	IF NOT #MovementActive THEN
	    FOR #i := 0 TO 12 DO
	        IF #ProductBuffer[#i].Active THEN
	            // Distance is oriented by DirectionSign:
	            //  - If DirectionSign = +1: Distance = Encoder - Start  (forward positive)
	            //  - If DirectionSign = -1: Distance = Start   - Encoder (forward negative)
	            #Distance := #DirectionSign * (#EncoderPosition - #ProductBuffer[#i].StartPosition);
	            
	            IF #Distance >= #TriggerDistance THEN
	                #TriggerMovement := TRUE;
	                #MovementActive := TRUE;
	                #ProductBuffer[#i].Active := FALSE;
	                EXIT;
	            END_IF;
	        END_IF;
	    END_FOR;
	END_IF;
	
	
	// 4️⃣ Wacht op feedback om beweging af te ronden
	IF #MovementActive AND #TriggerFeedback THEN
	    #TriggerMovement := FALSE;
	    #MovementActive := FALSE;
	END_IF;
	
END_FUNCTION_BLOCK

FUNCTION_BLOCK "BlowOff_Timer"
{ S7_Optimized_Access := 'FALSE' }
VERSION : 0.1
   VAR_INPUT 
      Enable : Bool;
      CycleTime : Time;
      PulseDuration : Time;
      NowTime : Time;
   END_VAR

   VAR_OUTPUT 
      Q_Pulse : Bool;
   END_VAR

   VAR 
      CycleTimer {InstructionName := 'TON'; LibVersion := '1.0'; S7_SetPoint := 'False'} : TON;
      PulseTimer {InstructionName := 'TON'; LibVersion := '1.0'; S7_SetPoint := 'False'} : TON;
      State { S7_SetPoint := 'True'} : Int;
      S_PEXT : Int;
   END_VAR

   VAR_TEMP 
      PulseActive : Bool;
      StartPulse : Bool;
      TriggerPulse : Bool;
      PulseBusy : Bool;
      DummyWord : Word;
      DummyWord2 : Bool;
      T1 : Int;
      PulseStartTime : Time;
      LastPulseEndTime : Time;
      LastPulseTime : Time;
   END_VAR


BEGIN
	// Logica
	IF #Enable THEN
	    // Start cyclische timer
	    #CycleTimer(IN := TRUE,
	                PT := #CycleTime);
	    
	    IF #CycleTimer.Q THEN
	        // Start puls-timer als cyclus voorbij is
	        #PulseTimer(IN := TRUE,
	                    PT := #PulseDuration);
	        
	        // Reset de CycleTimer voor de volgende cyclus
	        #CycleTimer(IN := FALSE,
	                    PT := #CycleTime);
	    END_IF;
	    
	    // Puls-timer logica
	    IF #PulseTimer.IN THEN
	        #Q_Pulse := TRUE;
	        
	        IF #PulseTimer.Q THEN
	            // Puls voorbij, pulse output uit
	            #PulseTimer(IN := FALSE,
	                        PT := #PulseDuration);
	            #Q_Pulse := FALSE;
	        END_IF;
	    ELSE
	        #Q_Pulse := FALSE;
	    END_IF;
	    
	ELSE
	    // Alles resetten bij disable
	    #CycleTimer(IN := FALSE,
	                PT := #CycleTime);
	    #PulseTimer(IN := FALSE,
	                PT := #PulseDuration);
	    #Q_Pulse := FALSE;
	END_IF;
	
END_FUNCTION_BLOCK

FUNCTION "4 - Prog. 2" : Void   // FC2, LAD
TITLE = System Program 2
VERSION : 0.1
// stored: AutoNumber true, IsIECCheckEnabled false, UDAEnableTagReadback false
   VAR_TEMP
      Retourband_Delayed : Bool;
      BlowOffTimer : Bool;
      Democoil : Bool;
      StartBlowOff : Bool;
      Pos2_Done : Bool;
      BlowOff_Activated : Bool;
      AandrukCilindersOut : Bool;
      Move2Busy : Bool;
      ProductBehindWals : Bool;
      SR_Move2 : Bool;
      Move1Busy : Bool;
   END_VAR
   VAR_TEMP   // added for the SCL form of the ladder/FBD networks
      _w1 : Bool;
   END_VAR
BEGIN

REGION Network 1: Close 1 Magazine Hole (cilinder)
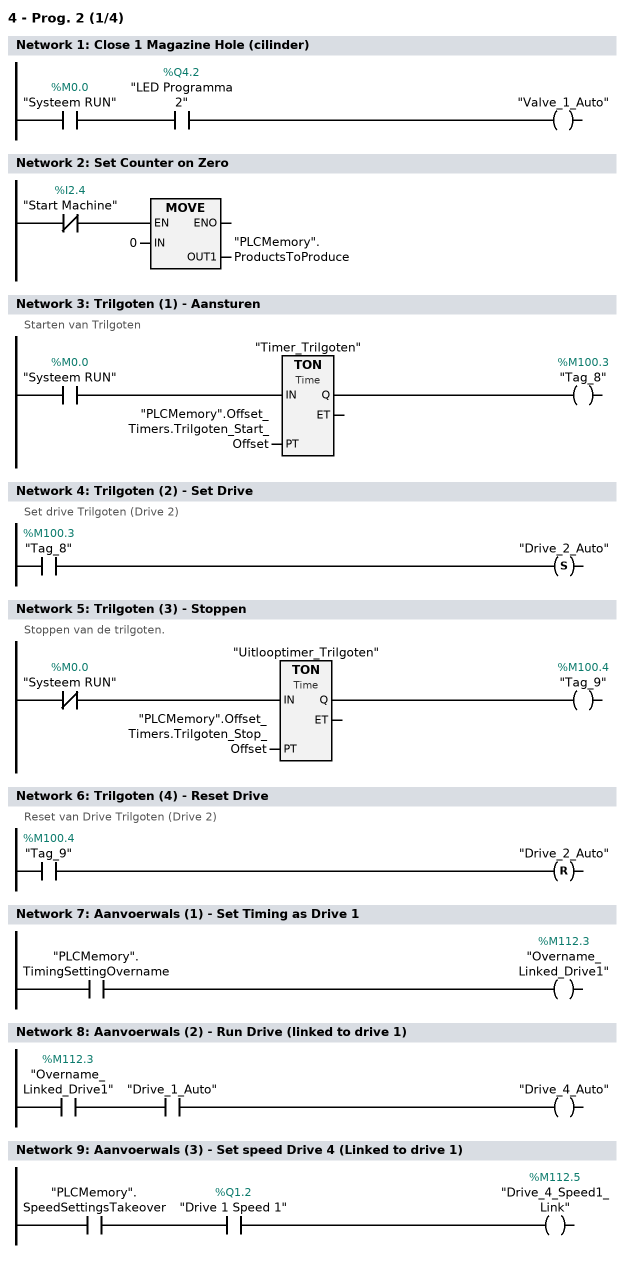
   RUNG wire#powerrail
      Contact( "Systeem RUN" )
      Contact( "LED Programma 2" )
      Coil( "Valve_1_Auto" )
   END_RUNG
   // the same network as SCL:
   "Valve_1_Auto" := "Systeem RUN" AND "LED Programma 2";
END_REGION

REGION Network 2: Set Counter on Zero
   RUNG wire#powerrail
      I_Contact( "Start Machine" )
      { S7_GenerateENO := "TRUE" } Move(in := 0, out1 => "PLCMemory".ProductsToProduce)
   END_RUNG
   // the same network as SCL:
   IF NOT "Start Machine" THEN "PLCMemory".ProductsToProduce := 0; END_IF;
END_REGION

REGION Network 3: Trilgoten (1) - Aansturen
   // Starten van Trilgoten
   RUNG wire#powerrail
      Contact( "Systeem RUN" )
      { S7_Templates := "time_type := Time" } "Timer_Trilgoten".TON(pt := "PLCMemory".Offset_Timers.Trilgoten_Start_Offset, et =>)
      Coil( "Tag_8" )
   END_RUNG
   // the same network as SCL:
   "Timer_Trilgoten".TON(IN := "Systeem RUN", PT := "PLCMemory".Offset_Timers.Trilgoten_Start_Offset);
   "Tag_8" := "Timer_Trilgoten".Q;
END_REGION

REGION Network 4: Trilgoten (2) - Set Drive
   // Set drive Trilgoten (Drive 2)
   RUNG wire#powerrail
      Contact( "Tag_8" )
      S_Coil( "Drive_2_Auto" )
   END_RUNG
   // the same network as SCL:
   IF "Tag_8" THEN "Drive_2_Auto" := TRUE; END_IF;
END_REGION

REGION Network 5: Trilgoten (3) - Stoppen
   // Stoppen van de trilgoten.
   RUNG wire#powerrail
      I_Contact( "Systeem RUN" )
      { S7_Templates := "time_type := Time" } "Uitlooptimer_Trilgoten".TON(pt := "PLCMemory".Offset_Timers.Trilgoten_Stop_Offset, et =>)
      Coil( "Tag_9" )
   END_RUNG
   // the same network as SCL:
   "Uitlooptimer_Trilgoten".TON(IN := NOT "Systeem RUN", PT := "PLCMemory".Offset_Timers.Trilgoten_Stop_Offset);
   "Tag_9" := "Uitlooptimer_Trilgoten".Q;
END_REGION

REGION Network 6: Trilgoten (4) - Reset Drive
   // Reset van Drive Trilgoten (Drive 2)
   RUNG wire#powerrail
      Contact( "Tag_9" )
      R_Coil( "Drive_2_Auto" )
   END_RUNG
   // the same network as SCL:
   IF "Tag_9" THEN "Drive_2_Auto" := FALSE; END_IF;
END_REGION

REGION Network 7: Aanvoerwals (1) - Set Timing as Drive 1
   RUNG wire#powerrail
      Contact( "PLCMemory".TimingSettingOvername )
      Coil( "Overname_Linked_Drive1" )
   END_RUNG
   // the same network as SCL:
   "Overname_Linked_Drive1" := "PLCMemory".TimingSettingOvername;
END_REGION

REGION Network 8: Aanvoerwals (2) - Run Drive (linked to drive 1)
   RUNG wire#powerrail
      Contact( "Overname_Linked_Drive1" )
      Contact( "Drive_1_Auto" )
      Coil( "Drive_4_Auto" )
   END_RUNG
   // the same network as SCL:
   "Drive_4_Auto" := "Overname_Linked_Drive1" AND "Drive_1_Auto";
END_REGION

REGION Network 9: Aanvoerwals (3) - Set speed Drive 4 (Linked to drive 1)
   RUNG wire#powerrail
      Contact( "PLCMemory".SpeedSettingsTakeover )
      Contact( "Drive 1 Speed 1" )
      Coil( "Drive_4_Speed1_Link" )
   END_RUNG
   // the same network as SCL:
   "Drive_4_Speed1_Link" := "PLCMemory".SpeedSettingsTakeover AND "Drive 1 Speed 1";
END_REGION

REGION Network 10: Aanvoerwals (4) - Set alternative Speed 1
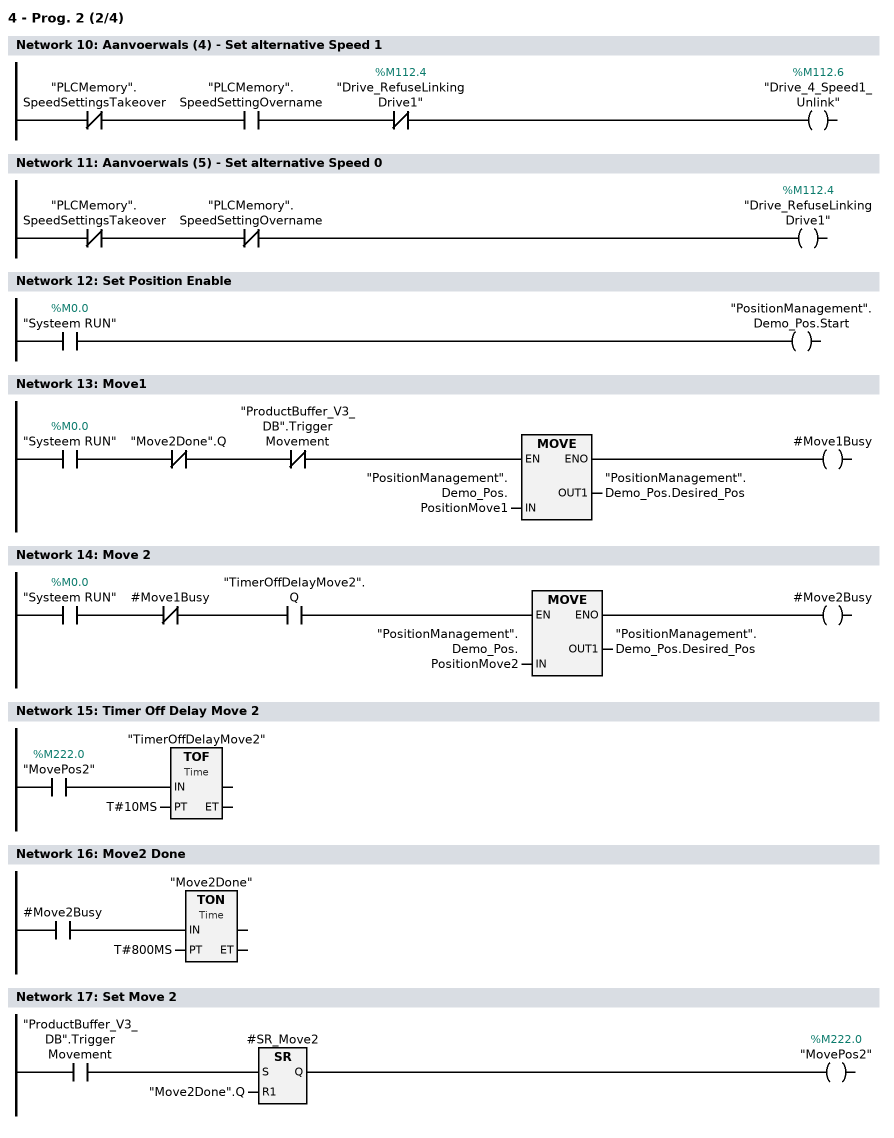
   RUNG wire#powerrail
      I_Contact( "PLCMemory".SpeedSettingsTakeover )
      Contact( "PLCMemory".SpeedSettingOvername )
      I_Contact( "Drive_RefuseLinkingDrive1" )
      Coil( "Drive_4_Speed1_Unlink" )
   END_RUNG
   // the same network as SCL:
   "Drive_4_Speed1_Unlink" := NOT "PLCMemory".SpeedSettingsTakeover AND "PLCMemory".SpeedSettingOvername AND NOT "Drive_RefuseLinkingDrive1";
END_REGION

REGION Network 11: Aanvoerwals (5) - Set alternative Speed 0
   RUNG wire#powerrail
      I_Contact( "PLCMemory".SpeedSettingsTakeover )
      I_Contact( "PLCMemory".SpeedSettingOvername )
      Coil( "Drive_RefuseLinkingDrive1" )
   END_RUNG
   // the same network as SCL:
   "Drive_RefuseLinkingDrive1" := NOT "PLCMemory".SpeedSettingsTakeover AND NOT "PLCMemory".SpeedSettingOvername;
END_REGION

REGION Network 12: Set Position Enable
   RUNG wire#powerrail
      Contact( "Systeem RUN" )
      Coil( "PositionManagement".Demo_Pos.Start )
   END_RUNG
   // the same network as SCL:
   "PositionManagement".Demo_Pos.Start := "Systeem RUN";
END_REGION

REGION Network 13: Move1
   RUNG wire#powerrail
      Contact( "Systeem RUN" )
      I_Contact( "Move2Done".Q )
      I_Contact( "ProductBuffer_V3_DB".TriggerMovement )
      { S7_GenerateENO := "TRUE" } Move(in := "PositionManagement".Demo_Pos.PositionMove1, out1 => "PositionManagement".Demo_Pos.Desired_Pos)
      Coil( #Move1Busy )
   END_RUNG
   // the same network as SCL:
   // ENO of a box is taken as its EN; it also drops when the box reports an error
   #_w1 := "Systeem RUN" AND NOT "Move2Done".Q AND NOT "ProductBuffer_V3_DB".TriggerMovement;
   IF #_w1 THEN
       "PositionManagement".Demo_Pos.Desired_Pos := "PositionManagement".Demo_Pos.PositionMove1;
   END_IF;
   #Move1Busy := #_w1;
END_REGION

REGION Network 14: Move 2
   RUNG wire#powerrail
      Contact( "Systeem RUN" )
      I_Contact( #Move1Busy )
      Contact( "TimerOffDelayMove2".Q )
      { S7_GenerateENO := "TRUE" } Move(in := "PositionManagement".Demo_Pos.PositionMove2, out1 => "PositionManagement".Demo_Pos.Desired_Pos)
      Coil( #Move2Busy )
   END_RUNG
   // the same network as SCL:
   // ENO of a box is taken as its EN; it also drops when the box reports an error
   #_w1 := "Systeem RUN" AND NOT #Move1Busy AND "TimerOffDelayMove2".Q;
   IF #_w1 THEN
       "PositionManagement".Demo_Pos.Desired_Pos := "PositionManagement".Demo_Pos.PositionMove2;
   END_IF;
   #Move2Busy := #_w1;
END_REGION

REGION Network 15: Timer Off Delay Move 2
   RUNG wire#powerrail
      Contact( "MovePos2" )
      { S7_Templates := "time_type := Time" } "TimerOffDelayMove2".TOF(pt := T#10MS, et =>)
   END_RUNG
   // the same network as SCL:
   "TimerOffDelayMove2".TOF(IN := "MovePos2", PT := T#10MS);
END_REGION

REGION Network 16: Move2 Done
   RUNG wire#powerrail
      Contact( #Move2Busy )
      { S7_Templates := "time_type := Time" } "Move2Done".TON(pt := T#800MS, et =>)
   END_RUNG
   // the same network as SCL:
   "Move2Done".TON(IN := #Move2Busy, PT := T#800MS);
END_REGION

REGION Network 17: Set Move 2
   RUNG wire#powerrail
      Contact( "ProductBuffer_V3_DB".TriggerMovement )
      S_SR(operand := #SR_Move2, r1 := "Move2Done".Q)
      Coil( "MovePos2" )
   END_RUNG
   // the same network as SCL:
   IF "ProductBuffer_V3_DB".TriggerMovement THEN
       #SR_Move2 := TRUE;   // SR flip-flop
   END_IF;
   IF "Move2Done".Q THEN #SR_Move2 := FALSE; END_IF;
   "MovePos2" := #SR_Move2;
END_REGION

REGION Network 18: Set Product Behind WalsOld V2.
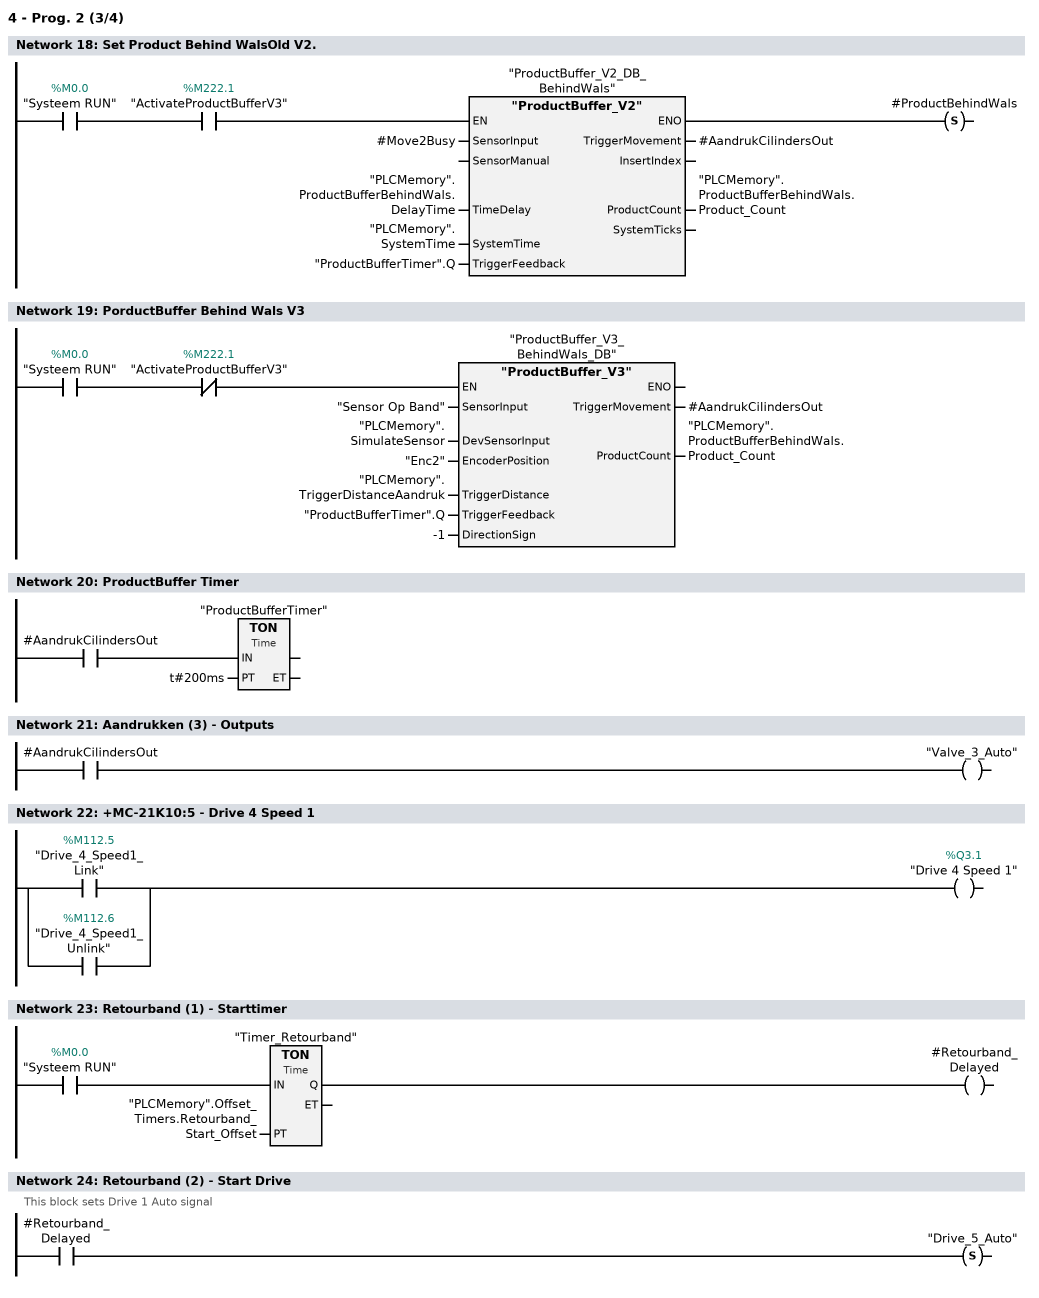
   RUNG wire#powerrail
      Contact( "Systeem RUN" )
      Contact( "ActivateProductBufferV3" )
      "ProductBuffer_V2_DB_BehindWals"(SensorInput := #Move2Busy, SensorManual :=, TimeDelay := "PLCMemory".ProductBufferBehindWals.DelayTime, SystemTime := "PLCMemory".SystemTime, TriggerFeedback := "ProductBufferTimer".Q, TriggerMovement => #AandrukCilindersOut, InsertIndex =>, ProductCount => "PLCMemory".ProductBufferBehindWals.Product_Count, SystemTicks =>)
      S_Coil( #ProductBehindWals )
   END_RUNG
   // the same network as SCL:
   "ProductBuffer_V2_DB_BehindWals"(EN := "Systeem RUN" AND "ActivateProductBufferV3",   // "ProductBuffer_V2"
                           SensorInput := #Move2Busy,
                           TimeDelay := "PLCMemory".ProductBufferBehindWals.DelayTime,
                           SystemTime := "PLCMemory".SystemTime,
                           TriggerFeedback := "ProductBufferTimer".Q,
                           TriggerMovement => #AandrukCilindersOut,
                           ProductCount => "PLCMemory".ProductBufferBehindWals.Product_Count,
                           ENO => #_w1);
   IF #_w1 THEN #ProductBehindWals := TRUE; END_IF;
END_REGION

REGION Network 19: PorductBuffer Behind Wals V3
   RUNG wire#powerrail
      Contact( "Systeem RUN" )
      I_Contact( "ActivateProductBufferV3" )
      "ProductBuffer_V3_BehindWals_DB"(SensorInput := "Sensor Op Band", DevSensorInput := "PLCMemory".SimulateSensor, EncoderPosition := "Enc2", TriggerDistance := "PLCMemory".TriggerDistanceAandruk, TriggerFeedback := "ProductBufferTimer".Q, DirectionSign := -1, TriggerMovement => #AandrukCilindersOut, ProductCount => "PLCMemory".ProductBufferBehindWals.Product_Count)
   END_RUNG
   // the same network as SCL:
   IF "Systeem RUN" AND NOT "ActivateProductBufferV3" THEN
       "ProductBuffer_V3_BehindWals_DB"(SensorInput := "Sensor Op Band",   // "ProductBuffer_V3"
                               DevSensorInput := "PLCMemory".SimulateSensor,
                               EncoderPosition := "Enc2",
                               TriggerDistance := "PLCMemory".TriggerDistanceAandruk,
                               TriggerFeedback := "ProductBufferTimer".Q,
                               DirectionSign := -1,
                               TriggerMovement => #AandrukCilindersOut,
                               ProductCount => "PLCMemory".ProductBufferBehindWals.Product_Count);
   END_IF;
END_REGION

REGION Network 20: ProductBuffer Timer
   RUNG wire#powerrail
      Contact( #AandrukCilindersOut )
      { S7_Templates := "time_type := Time" } "ProductBufferTimer".TON(pt := t#200ms, et =>)
   END_RUNG
   // the same network as SCL:
   "ProductBufferTimer".TON(IN := #AandrukCilindersOut, PT := t#200ms);
END_REGION

REGION Network 21: Aandrukken (3) - Outputs
   RUNG wire#powerrail
      Contact( #AandrukCilindersOut )
      Coil( "Valve_3_Auto" )
   END_RUNG
   // the same network as SCL:
   "Valve_3_Auto" := #AandrukCilindersOut;
END_REGION

REGION Network 22: +MC-21K10:5 - Drive 4 Speed 1
   RUNG wire#powerrail
      Contact( "Drive_4_Speed1_Link" )
      wire#w1
      Coil( "Drive 4 Speed 1" )
   END_RUNG
   RUNG wire#powerrail
      Contact( "Drive_4_Speed1_Unlink" )
   END_RUNG wire#w1
   // the same network as SCL:
   "Drive 4 Speed 1" := "Drive_4_Speed1_Link" OR "Drive_4_Speed1_Unlink";
END_REGION

REGION Network 23: Retourband (1) - Starttimer
   RUNG wire#powerrail
      Contact( "Systeem RUN" )
      { S7_Templates := "time_type := Time" } "Timer_Retourband".TON(pt := "PLCMemory".Offset_Timers.Retourband_Start_Offset, et =>)
      Coil( #Retourband_Delayed )
   END_RUNG
   // the same network as SCL:
   "Timer_Retourband".TON(IN := "Systeem RUN", PT := "PLCMemory".Offset_Timers.Retourband_Start_Offset);
   #Retourband_Delayed := "Timer_Retourband".Q;
END_REGION

REGION Network 24: Retourband (2) - Start Drive
   // This block sets Drive 1 Auto signal
   RUNG wire#powerrail
      Contact( #Retourband_Delayed )
      S_Coil( "Drive_5_Auto" )
   END_RUNG
   // the same network as SCL:
   IF #Retourband_Delayed THEN "Drive_5_Auto" := TRUE; END_IF;
END_REGION

REGION Network 25: Retourband (3) - Stop Drive
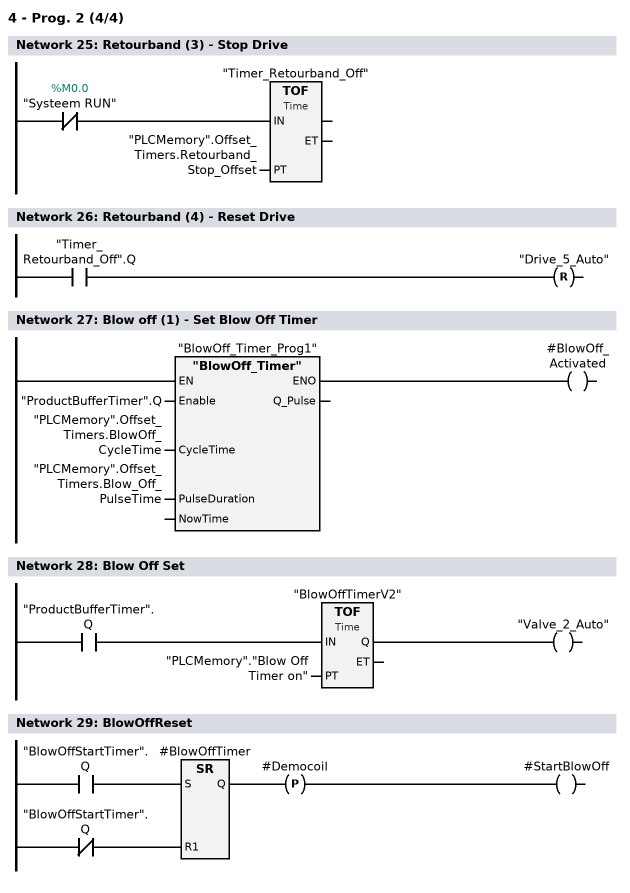
   RUNG wire#powerrail
      I_Contact( "Systeem RUN" )
      { S7_Templates := "time_type := Time" } "Timer_Retourband_Off".TOF(pt := "PLCMemory".Offset_Timers.Retourband_Stop_Offset, et =>)
   END_RUNG
   // the same network as SCL:
   "Timer_Retourband_Off".TOF(IN := NOT "Systeem RUN", PT := "PLCMemory".Offset_Timers.Retourband_Stop_Offset);
END_REGION

REGION Network 26: Retourband (4) - Reset Drive
   RUNG wire#powerrail
      Contact( "Timer_Retourband_Off".Q )
      R_Coil( "Drive_5_Auto" )
   END_RUNG
   // the same network as SCL:
   IF "Timer_Retourband_Off".Q THEN "Drive_5_Auto" := FALSE; END_IF;
END_REGION

REGION Network 27: Blow off (1) - Set Blow Off Timer
   RUNG wire#powerrail
      "BlowOff_Timer_Prog1"(Enable := "ProductBufferTimer".Q, CycleTime := "PLCMemory".Offset_Timers.BlowOff_CycleTime, PulseDuration := "PLCMemory".Offset_Timers.Blow_Off_PulseTime, NowTime :=, Q_Pulse =>)
      Coil( #BlowOff_Activated )
   END_RUNG
   // the same network as SCL:
   "BlowOff_Timer_Prog1"(Enable := "ProductBufferTimer".Q,   // "BlowOff_Timer"
                         CycleTime := "PLCMemory".Offset_Timers.BlowOff_CycleTime,
                         PulseDuration := "PLCMemory".Offset_Timers.Blow_Off_PulseTime,
                         ENO => #_w1);
   #BlowOff_Activated := #_w1;
END_REGION

REGION Network 28: Blow Off Set
   RUNG wire#powerrail
      Contact( "ProductBufferTimer".Q )
      { S7_Templates := "time_type := Time" } "BlowOffTimerV2".TOF(pt := "PLCMemory"."Blow Off Timer on", et =>)
      Coil( "Valve_2_Auto" )
   END_RUNG
   // the same network as SCL:
   "BlowOffTimerV2".TOF(IN := "ProductBufferTimer".Q, PT := "PLCMemory"."Blow Off Timer on");
   "Valve_2_Auto" := "BlowOffTimerV2".Q;
END_REGION

REGION Network 29: BlowOffReset
   RUNG wire#powerrail
      Contact( "BlowOffStartTimer".Q )
      S_SR(operand := #BlowOffTimer, r1 := wire#w1)
      P_Trig( #Democoil )
      Coil( #StartBlowOff )
   END_RUNG
   RUNG wire#powerrail
      I_Contact( "BlowOffStartTimer".Q )
   END_RUNG wire#w1
   // the same network as SCL:
   IF "BlowOffStartTimer".Q THEN
       #BlowOffTimer := TRUE;   // SR flip-flop
   END_IF;
   IF NOT "BlowOffStartTimer".Q THEN #BlowOffTimer := FALSE; END_IF;
   #_w1 := #BlowOffTimer AND NOT #Democoil;   // rising edge
   #Democoil := #BlowOffTimer;
   #StartBlowOff := #_w1;
END_REGION
END_FUNCTION

FUNCTION "5 - Prog. 3" : Void   // FC3, LAD
TITLE = System Program 3
VERSION : 0.1
// stored: AutoNumber true, IsIECCheckEnabled false, UDAEnableTagReadback false
   VAR_TEMP
      BlowOffTimer : Bool;
      Democoil : Bool;
      StartBlowOff : Bool;
      Pos2_Done : Bool;
      BlowOff_Activated : Bool;
      Retourband_Delayed : Bool;
      AandrukCilindersOut : Bool;
      Move2Busy : Bool;
      ProductBehindWals : Bool;
      SR_Move2 : Bool;
      Move1Busy : Bool;
   END_VAR
   VAR_TEMP   // added for the SCL form of the ladder/FBD networks
      _w1 : Bool;
   END_VAR
BEGIN

REGION Network 1: Close 1 Magazine Hole (cilinder)
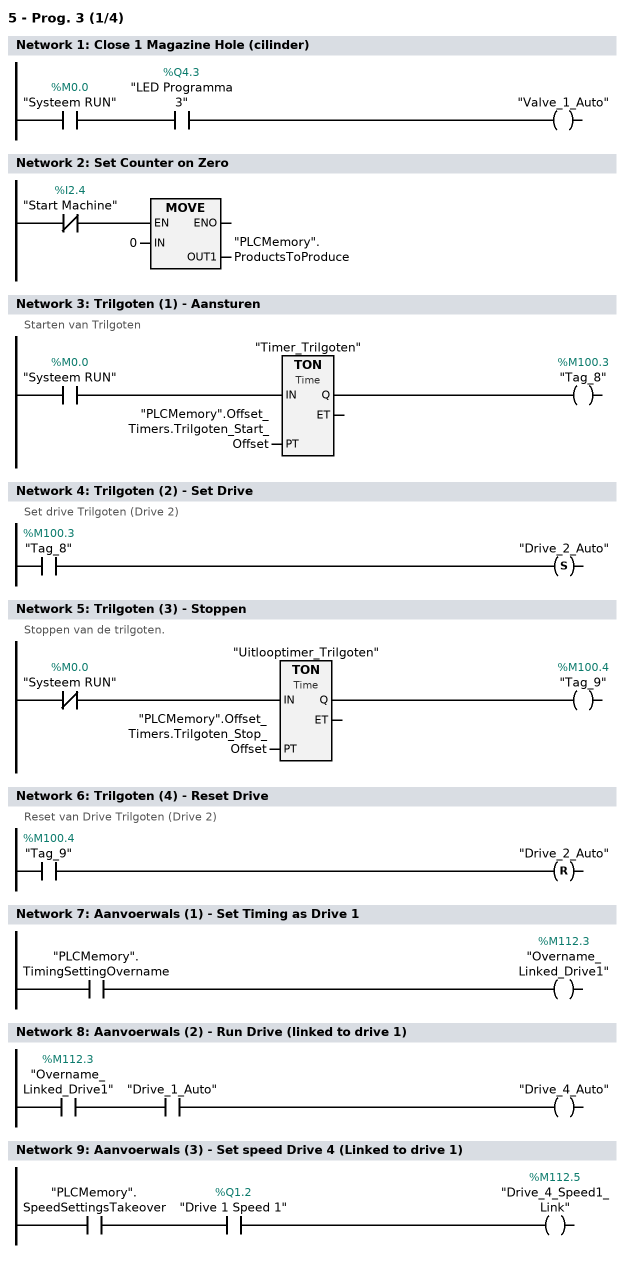
   RUNG wire#powerrail
      Contact( "Systeem RUN" )
      Contact( "LED Programma 3" )
      Coil( "Valve_1_Auto" )
   END_RUNG
   // the same network as SCL:
   "Valve_1_Auto" := "Systeem RUN" AND "LED Programma 3";
END_REGION

REGION Network 2: Set Counter on Zero
   RUNG wire#powerrail
      I_Contact( "Start Machine" )
      { S7_GenerateENO := "TRUE" } Move(in := 0, out1 => "PLCMemory".ProductsToProduce)
   END_RUNG
   // the same network as SCL:
   IF NOT "Start Machine" THEN "PLCMemory".ProductsToProduce := 0; END_IF;
END_REGION

REGION Network 3: Trilgoten (1) - Aansturen
   // Starten van Trilgoten
   RUNG wire#powerrail
      Contact( "Systeem RUN" )
      { S7_Templates := "time_type := Time" } "Timer_Trilgoten".TON(pt := "PLCMemory".Offset_Timers.Trilgoten_Start_Offset, et =>)
      Coil( "Tag_8" )
   END_RUNG
   // the same network as SCL:
   "Timer_Trilgoten".TON(IN := "Systeem RUN", PT := "PLCMemory".Offset_Timers.Trilgoten_Start_Offset);
   "Tag_8" := "Timer_Trilgoten".Q;
END_REGION

REGION Network 4: Trilgoten (2) - Set Drive
   // Set drive Trilgoten (Drive 2)
   RUNG wire#powerrail
      Contact( "Tag_8" )
      S_Coil( "Drive_2_Auto" )
   END_RUNG
   // the same network as SCL:
   IF "Tag_8" THEN "Drive_2_Auto" := TRUE; END_IF;
END_REGION

REGION Network 5: Trilgoten (3) - Stoppen
   // Stoppen van de trilgoten.
   RUNG wire#powerrail
      I_Contact( "Systeem RUN" )
      { S7_Templates := "time_type := Time" } "Uitlooptimer_Trilgoten".TON(pt := "PLCMemory".Offset_Timers.Trilgoten_Stop_Offset, et =>)
      Coil( "Tag_9" )
   END_RUNG
   // the same network as SCL:
   "Uitlooptimer_Trilgoten".TON(IN := NOT "Systeem RUN", PT := "PLCMemory".Offset_Timers.Trilgoten_Stop_Offset);
   "Tag_9" := "Uitlooptimer_Trilgoten".Q;
END_REGION

REGION Network 6: Trilgoten (4) - Reset Drive
   // Reset van Drive Trilgoten (Drive 2)
   RUNG wire#powerrail
      Contact( "Tag_9" )
      R_Coil( "Drive_2_Auto" )
   END_RUNG
   // the same network as SCL:
   IF "Tag_9" THEN "Drive_2_Auto" := FALSE; END_IF;
END_REGION

REGION Network 7: Aanvoerwals (1) - Set Timing as Drive 1
   RUNG wire#powerrail
      Contact( "PLCMemory".TimingSettingOvername )
      Coil( "Overname_Linked_Drive1" )
   END_RUNG
   // the same network as SCL:
   "Overname_Linked_Drive1" := "PLCMemory".TimingSettingOvername;
END_REGION

REGION Network 8: Aanvoerwals (2) - Run Drive (linked to drive 1)
   RUNG wire#powerrail
      Contact( "Overname_Linked_Drive1" )
      Contact( "Drive_1_Auto" )
      Coil( "Drive_4_Auto" )
   END_RUNG
   // the same network as SCL:
   "Drive_4_Auto" := "Overname_Linked_Drive1" AND "Drive_1_Auto";
END_REGION

REGION Network 9: Aanvoerwals (3) - Set speed Drive 4 (Linked to drive 1)
   RUNG wire#powerrail
      Contact( "PLCMemory".SpeedSettingsTakeover )
      Contact( "Drive 1 Speed 1" )
      Coil( "Drive_4_Speed1_Link" )
   END_RUNG
   // the same network as SCL:
   "Drive_4_Speed1_Link" := "PLCMemory".SpeedSettingsTakeover AND "Drive 1 Speed 1";
END_REGION

REGION Network 10: Aanvoerwals (4) - Set alternative Speed 1
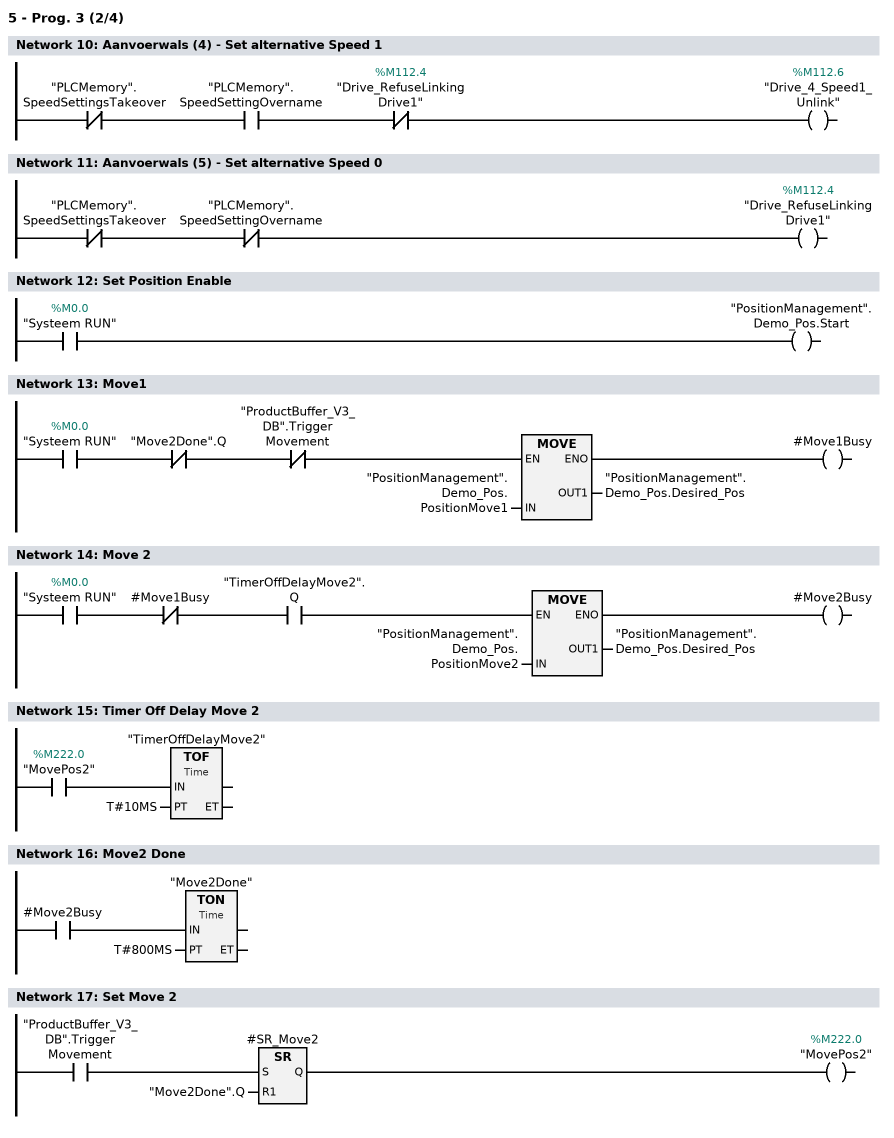
   RUNG wire#powerrail
      I_Contact( "PLCMemory".SpeedSettingsTakeover )
      Contact( "PLCMemory".SpeedSettingOvername )
      I_Contact( "Drive_RefuseLinkingDrive1" )
      Coil( "Drive_4_Speed1_Unlink" )
   END_RUNG
   // the same network as SCL:
   "Drive_4_Speed1_Unlink" := NOT "PLCMemory".SpeedSettingsTakeover AND "PLCMemory".SpeedSettingOvername AND NOT "Drive_RefuseLinkingDrive1";
END_REGION

REGION Network 11: Aanvoerwals (5) - Set alternative Speed 0
   RUNG wire#powerrail
      I_Contact( "PLCMemory".SpeedSettingsTakeover )
      I_Contact( "PLCMemory".SpeedSettingOvername )
      Coil( "Drive_RefuseLinkingDrive1" )
   END_RUNG
   // the same network as SCL:
   "Drive_RefuseLinkingDrive1" := NOT "PLCMemory".SpeedSettingsTakeover AND NOT "PLCMemory".SpeedSettingOvername;
END_REGION

REGION Network 12: Set Position Enable
   RUNG wire#powerrail
      Contact( "Systeem RUN" )
      Coil( "PositionManagement".Demo_Pos.Start )
   END_RUNG
   // the same network as SCL:
   "PositionManagement".Demo_Pos.Start := "Systeem RUN";
END_REGION

REGION Network 13: Move1
   RUNG wire#powerrail
      Contact( "Systeem RUN" )
      I_Contact( "Move2Done".Q )
      I_Contact( "ProductBuffer_V3_DB".TriggerMovement )
      { S7_GenerateENO := "TRUE" } Move(in := "PositionManagement".Demo_Pos.PositionMove1, out1 => "PositionManagement".Demo_Pos.Desired_Pos)
      Coil( #Move1Busy )
   END_RUNG
   // the same network as SCL:
   // ENO of a box is taken as its EN; it also drops when the box reports an error
   #_w1 := "Systeem RUN" AND NOT "Move2Done".Q AND NOT "ProductBuffer_V3_DB".TriggerMovement;
   IF #_w1 THEN
       "PositionManagement".Demo_Pos.Desired_Pos := "PositionManagement".Demo_Pos.PositionMove1;
   END_IF;
   #Move1Busy := #_w1;
END_REGION

REGION Network 14: Move 2
   RUNG wire#powerrail
      Contact( "Systeem RUN" )
      I_Contact( #Move1Busy )
      Contact( "TimerOffDelayMove2".Q )
      { S7_GenerateENO := "TRUE" } Move(in := "PositionManagement".Demo_Pos.PositionMove2, out1 => "PositionManagement".Demo_Pos.Desired_Pos)
      Coil( #Move2Busy )
   END_RUNG
   // the same network as SCL:
   // ENO of a box is taken as its EN; it also drops when the box reports an error
   #_w1 := "Systeem RUN" AND NOT #Move1Busy AND "TimerOffDelayMove2".Q;
   IF #_w1 THEN
       "PositionManagement".Demo_Pos.Desired_Pos := "PositionManagement".Demo_Pos.PositionMove2;
   END_IF;
   #Move2Busy := #_w1;
END_REGION

REGION Network 15: Timer Off Delay Move 2
   RUNG wire#powerrail
      Contact( "MovePos2" )
      { S7_Templates := "time_type := Time" } "TimerOffDelayMove2".TOF(pt := T#10MS, et =>)
   END_RUNG
   // the same network as SCL:
   "TimerOffDelayMove2".TOF(IN := "MovePos2", PT := T#10MS);
END_REGION

REGION Network 16: Move2 Done
   RUNG wire#powerrail
      Contact( #Move2Busy )
      { S7_Templates := "time_type := Time" } "Move2Done".TON(pt := T#800MS, et =>)
   END_RUNG
   // the same network as SCL:
   "Move2Done".TON(IN := #Move2Busy, PT := T#800MS);
END_REGION

REGION Network 17: Set Move 2
   RUNG wire#powerrail
      Contact( "ProductBuffer_V3_DB".TriggerMovement )
      S_SR(operand := #SR_Move2, r1 := "Move2Done".Q)
      Coil( "MovePos2" )
   END_RUNG
   // the same network as SCL:
   IF "ProductBuffer_V3_DB".TriggerMovement THEN
       #SR_Move2 := TRUE;   // SR flip-flop
   END_IF;
   IF "Move2Done".Q THEN #SR_Move2 := FALSE; END_IF;
   "MovePos2" := #SR_Move2;
END_REGION

REGION Network 18: Set Product Behind WalsOld V2.
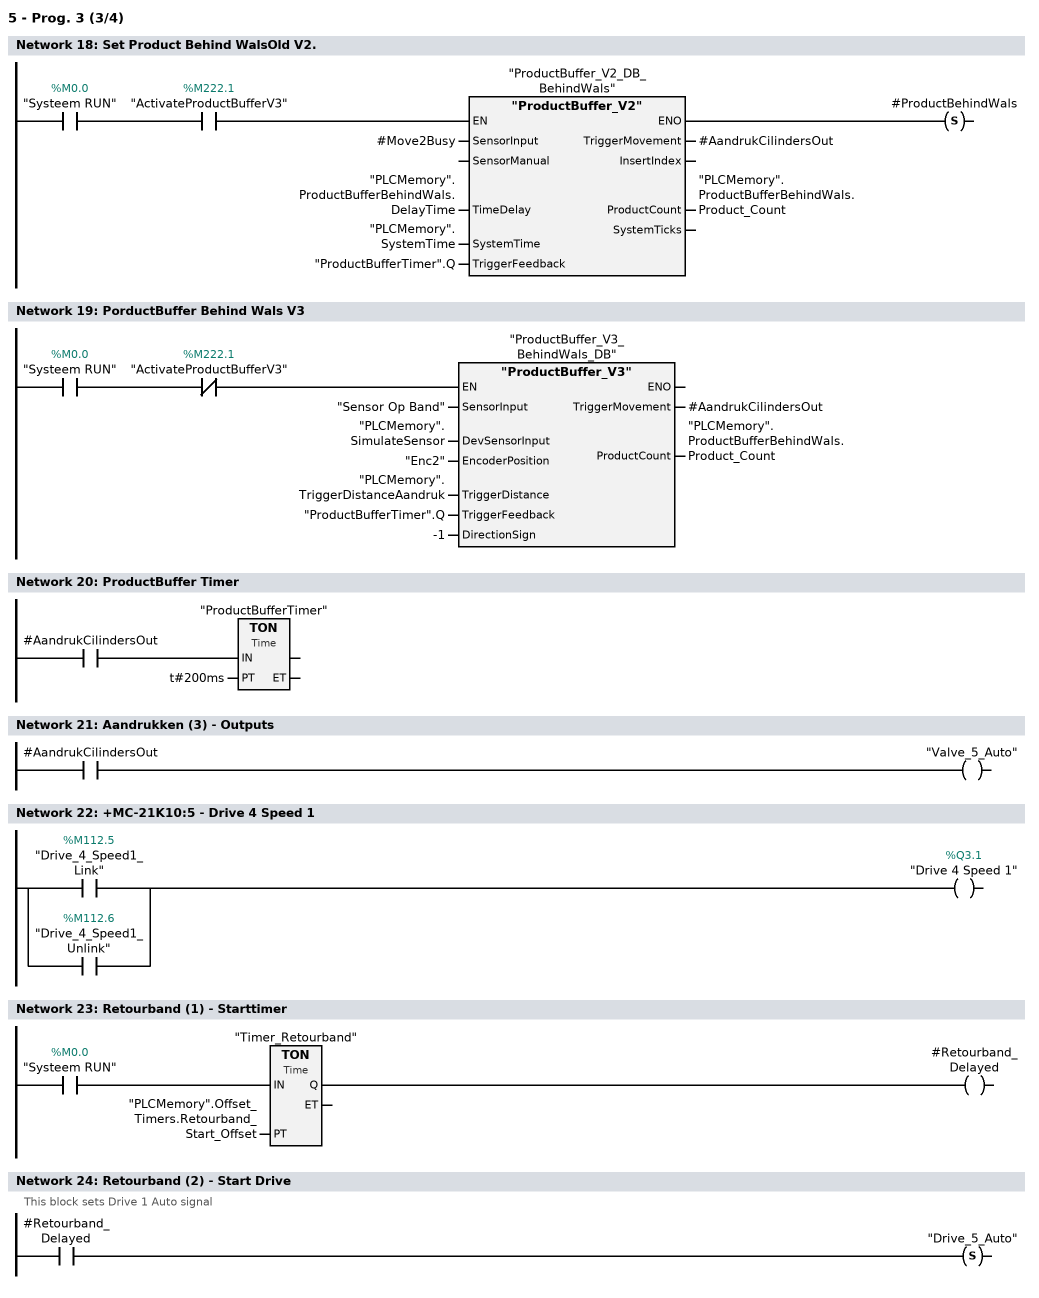
   RUNG wire#powerrail
      Contact( "Systeem RUN" )
      Contact( "ActivateProductBufferV3" )
      "ProductBuffer_V2_DB_BehindWals"(SensorInput := #Move2Busy, SensorManual :=, TimeDelay := "PLCMemory".ProductBufferBehindWals.DelayTime, SystemTime := "PLCMemory".SystemTime, TriggerFeedback := "ProductBufferTimer".Q, TriggerMovement => #AandrukCilindersOut, InsertIndex =>, ProductCount => "PLCMemory".ProductBufferBehindWals.Product_Count, SystemTicks =>)
      S_Coil( #ProductBehindWals )
   END_RUNG
   // the same network as SCL:
   "ProductBuffer_V2_DB_BehindWals"(EN := "Systeem RUN" AND "ActivateProductBufferV3",   // "ProductBuffer_V2"
                           SensorInput := #Move2Busy,
                           TimeDelay := "PLCMemory".ProductBufferBehindWals.DelayTime,
                           SystemTime := "PLCMemory".SystemTime,
                           TriggerFeedback := "ProductBufferTimer".Q,
                           TriggerMovement => #AandrukCilindersOut,
                           ProductCount => "PLCMemory".ProductBufferBehindWals.Product_Count,
                           ENO => #_w1);
   IF #_w1 THEN #ProductBehindWals := TRUE; END_IF;
END_REGION

REGION Network 19: PorductBuffer Behind Wals V3
   RUNG wire#powerrail
      Contact( "Systeem RUN" )
      I_Contact( "ActivateProductBufferV3" )
      "ProductBuffer_V3_BehindWals_DB"(SensorInput := "Sensor Op Band", DevSensorInput := "PLCMemory".SimulateSensor, EncoderPosition := "Enc2", TriggerDistance := "PLCMemory".TriggerDistanceAandruk, TriggerFeedback := "ProductBufferTimer".Q, DirectionSign := -1, TriggerMovement => #AandrukCilindersOut, ProductCount => "PLCMemory".ProductBufferBehindWals.Product_Count)
   END_RUNG
   // the same network as SCL:
   IF "Systeem RUN" AND NOT "ActivateProductBufferV3" THEN
       "ProductBuffer_V3_BehindWals_DB"(SensorInput := "Sensor Op Band",   // "ProductBuffer_V3"
                               DevSensorInput := "PLCMemory".SimulateSensor,
                               EncoderPosition := "Enc2",
                               TriggerDistance := "PLCMemory".TriggerDistanceAandruk,
                               TriggerFeedback := "ProductBufferTimer".Q,
                               DirectionSign := -1,
                               TriggerMovement => #AandrukCilindersOut,
                               ProductCount => "PLCMemory".ProductBufferBehindWals.Product_Count);
   END_IF;
END_REGION

REGION Network 20: ProductBuffer Timer
   RUNG wire#powerrail
      Contact( #AandrukCilindersOut )
      { S7_Templates := "time_type := Time" } "ProductBufferTimer".TON(pt := t#200ms, et =>)
   END_RUNG
   // the same network as SCL:
   "ProductBufferTimer".TON(IN := #AandrukCilindersOut, PT := t#200ms);
END_REGION

REGION Network 21: Aandrukken (3) - Outputs
   RUNG wire#powerrail
      Contact( #AandrukCilindersOut )
      Coil( "Valve_5_Auto" )
   END_RUNG
   // the same network as SCL:
   "Valve_5_Auto" := #AandrukCilindersOut;
END_REGION

REGION Network 22: +MC-21K10:5 - Drive 4 Speed 1
   RUNG wire#powerrail
      Contact( "Drive_4_Speed1_Link" )
      wire#w1
      Coil( "Drive 4 Speed 1" )
   END_RUNG
   RUNG wire#powerrail
      Contact( "Drive_4_Speed1_Unlink" )
   END_RUNG wire#w1
   // the same network as SCL:
   "Drive 4 Speed 1" := "Drive_4_Speed1_Link" OR "Drive_4_Speed1_Unlink";
END_REGION

REGION Network 23: Retourband (1) - Starttimer
   RUNG wire#powerrail
      Contact( "Systeem RUN" )
      { S7_Templates := "time_type := Time" } "Timer_Retourband".TON(pt := "PLCMemory".Offset_Timers.Retourband_Start_Offset, et =>)
      Coil( #Retourband_Delayed )
   END_RUNG
   // the same network as SCL:
   "Timer_Retourband".TON(IN := "Systeem RUN", PT := "PLCMemory".Offset_Timers.Retourband_Start_Offset);
   #Retourband_Delayed := "Timer_Retourband".Q;
END_REGION

REGION Network 24: Retourband (2) - Start Drive
   // This block sets Drive 1 Auto signal
   RUNG wire#powerrail
      Contact( #Retourband_Delayed )
      S_Coil( "Drive_5_Auto" )
   END_RUNG
   // the same network as SCL:
   IF #Retourband_Delayed THEN "Drive_5_Auto" := TRUE; END_IF;
END_REGION

REGION Network 25: Retourband (3) - Stop Drive
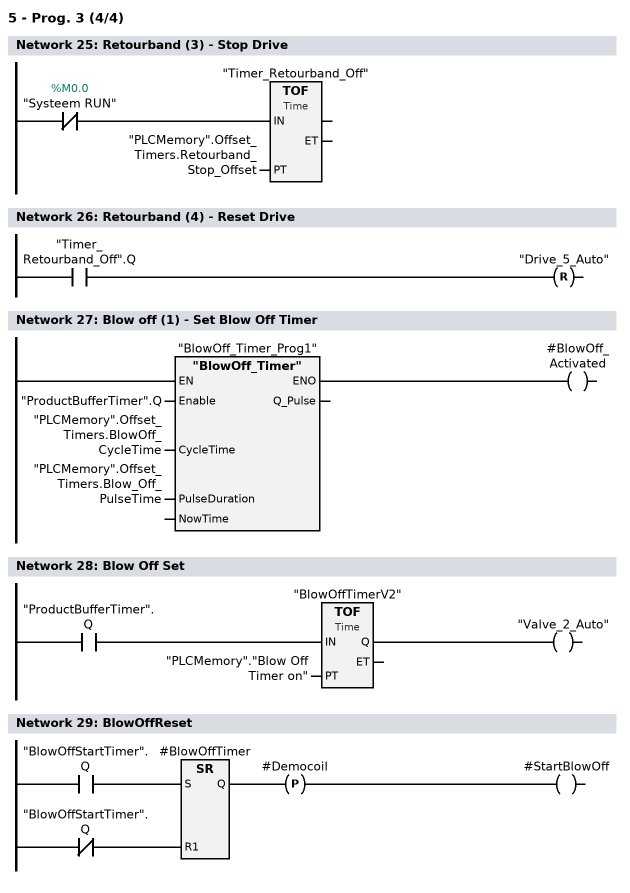
   RUNG wire#powerrail
      I_Contact( "Systeem RUN" )
      { S7_Templates := "time_type := Time" } "Timer_Retourband_Off".TOF(pt := "PLCMemory".Offset_Timers.Retourband_Stop_Offset, et =>)
   END_RUNG
   // the same network as SCL:
   "Timer_Retourband_Off".TOF(IN := NOT "Systeem RUN", PT := "PLCMemory".Offset_Timers.Retourband_Stop_Offset);
END_REGION

REGION Network 26: Retourband (4) - Reset Drive
   RUNG wire#powerrail
      Contact( "Timer_Retourband_Off".Q )
      R_Coil( "Drive_5_Auto" )
   END_RUNG
   // the same network as SCL:
   IF "Timer_Retourband_Off".Q THEN "Drive_5_Auto" := FALSE; END_IF;
END_REGION

REGION Network 27: Blow off (1) - Set Blow Off Timer
   RUNG wire#powerrail
      "BlowOff_Timer_Prog1"(Enable := "ProductBufferTimer".Q, CycleTime := "PLCMemory".Offset_Timers.BlowOff_CycleTime, PulseDuration := "PLCMemory".Offset_Timers.Blow_Off_PulseTime, NowTime :=, Q_Pulse =>)
      Coil( #BlowOff_Activated )
   END_RUNG
   // the same network as SCL:
   "BlowOff_Timer_Prog1"(Enable := "ProductBufferTimer".Q,   // "BlowOff_Timer"
                         CycleTime := "PLCMemory".Offset_Timers.BlowOff_CycleTime,
                         PulseDuration := "PLCMemory".Offset_Timers.Blow_Off_PulseTime,
                         ENO => #_w1);
   #BlowOff_Activated := #_w1;
END_REGION

REGION Network 28: Blow Off Set
   RUNG wire#powerrail
      Contact( "ProductBufferTimer".Q )
      { S7_Templates := "time_type := Time" } "BlowOffTimerV2".TOF(pt := "PLCMemory"."Blow Off Timer on", et =>)
      Coil( "Valve_2_Auto" )
   END_RUNG
   // the same network as SCL:
   "BlowOffTimerV2".TOF(IN := "ProductBufferTimer".Q, PT := "PLCMemory"."Blow Off Timer on");
   "Valve_2_Auto" := "BlowOffTimerV2".Q;
END_REGION

REGION Network 29: BlowOffReset
   RUNG wire#powerrail
      Contact( "BlowOffStartTimer".Q )
      S_SR(operand := #BlowOffTimer, r1 := wire#w1)
      P_Trig( #Democoil )
      Coil( #StartBlowOff )
   END_RUNG
   RUNG wire#powerrail
      I_Contact( "BlowOffStartTimer".Q )
   END_RUNG wire#w1
   // the same network as SCL:
   IF "BlowOffStartTimer".Q THEN
       #BlowOffTimer := TRUE;   // SR flip-flop
   END_IF;
   IF NOT "BlowOffStartTimer".Q THEN #BlowOffTimer := FALSE; END_IF;
   #_w1 := #BlowOffTimer AND NOT #Democoil;   // rising edge
   #Democoil := #BlowOffTimer;
   #StartBlowOff := #_w1;
END_REGION
END_FUNCTION

FUNCTION "1 - Outputs" : Void   // FC5, LAD
VERSION : 0.1
// This Function program is for operating the machine automatic and manual.
// stored: AutoNumber true, IsIECCheckEnabled false, UDAEnableTagReadback false
   VAR_TEMP
      Valve_2_Pulse : Bool;
      BlowOff_Activated : Bool;
      BlowOffManual : Bool;
      Pulse1 : Bool;
      Drive_1_ReferenceRun : Bool;
   END_VAR
   VAR_TEMP   // added for the SCL form of the ladder/FBD networks
      _w1 : Bool;
   END_VAR
BEGIN

REGION Network 1: Drive 1 - Control
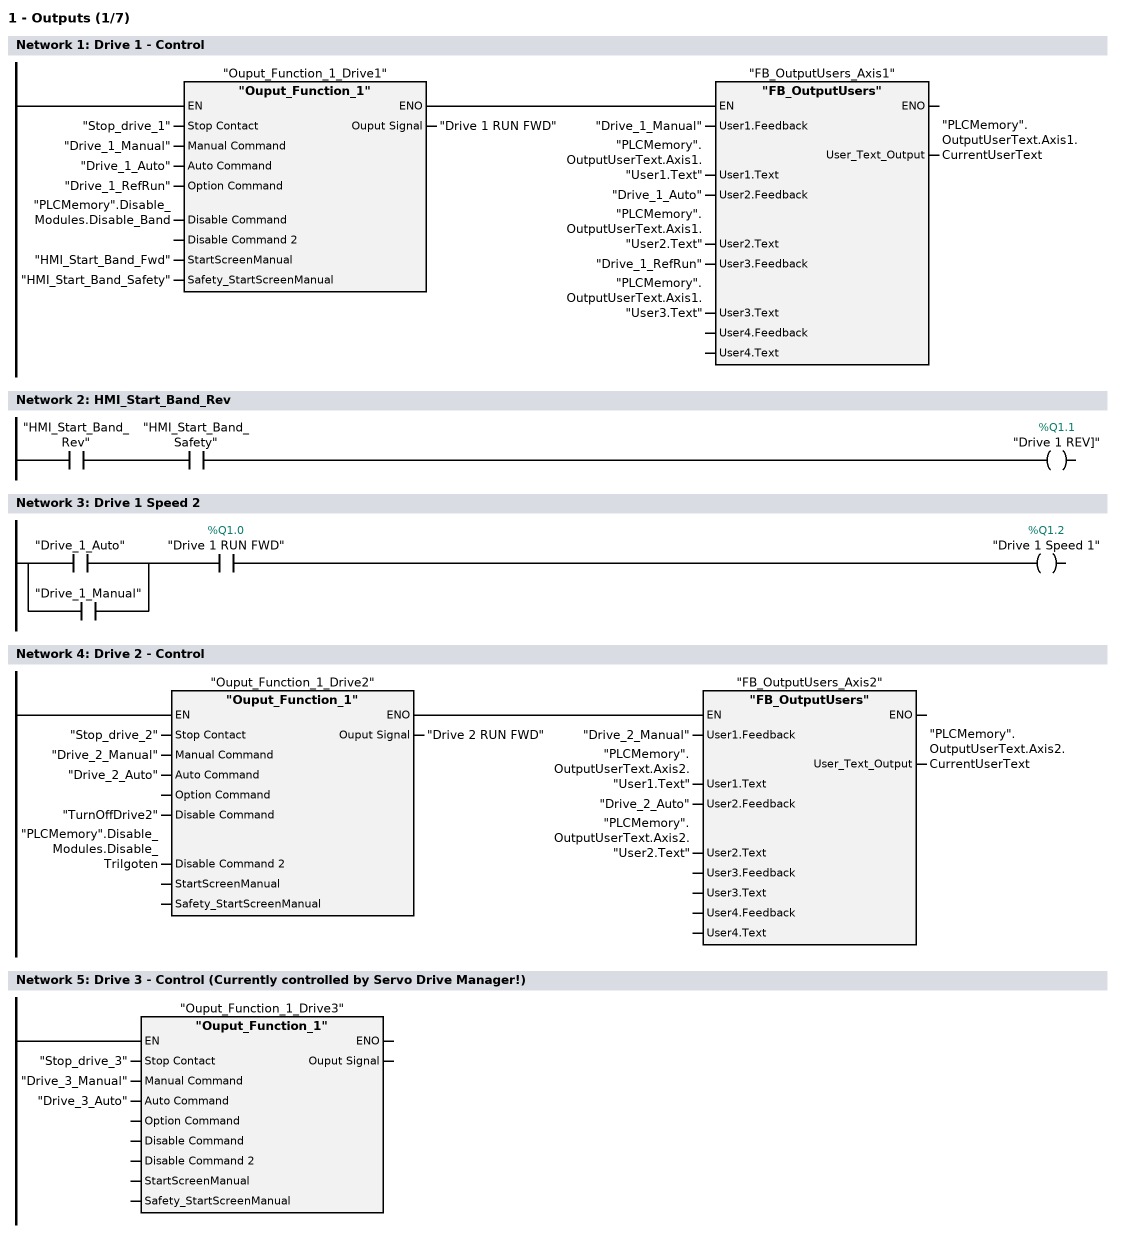
   RUNG wire#powerrail
      "Ouput_Function_1_Drive1"("Stop Contact" := "Stop_drive_1", "Manual Command" := "Drive_1_Manual", "Auto Command" := "Drive_1_Auto", "Option Command" := "Drive_1_RefRun", "Disable Command" := "PLCMemory".Disable_Modules.Disable_Band, "Disable Command 2" :=, StartScreenManual := "HMI_Start_Band_Fwd", Safety_StartScreenManual := "HMI_Start_Band_Safety", "Ouput Signal" => "Drive 1 RUN FWD")
      "FB_OutputUsers_Axis1"("User1.Feedback" := "Drive_1_Manual", "User1.Text" := "PLCMemory".OutputUserText.Axis1."User1.Text", "User2.Feedback" := "Drive_1_Auto", "User2.Text" := "PLCMemory".OutputUserText.Axis1."User2.Text", "User3.Feedback" := "Drive_1_RefRun", "User3.Text" := "PLCMemory".OutputUserText.Axis1."User3.Text", "User4.Feedback" :=, "User4.Text" :=, User_Text_Output => "PLCMemory".OutputUserText.Axis1.CurrentUserText)
   END_RUNG
   // the same network as SCL:
   "Ouput_Function_1_Drive1"("Stop Contact" := "Stop_drive_1",   // "Ouput_Function_1"
                           "Manual Command" := "Drive_1_Manual",
                           "Auto Command" := "Drive_1_Auto",
                           "Option Command" := "Drive_1_RefRun",
                           "Disable Command" := "PLCMemory".Disable_Modules.Disable_Band,
                           StartScreenManual := "HMI_Start_Band_Fwd",
                           Safety_StartScreenManual := "HMI_Start_Band_Safety",
                           "Ouput Signal" => "Drive 1 RUN FWD",
                           ENO => #_w1);
   IF #_w1 THEN
       "FB_OutputUsers_Axis1"("User1.Feedback" := "Drive_1_Manual",   // "FB_OutputUsers"
                              "User1.Text" := "PLCMemory".OutputUserText.Axis1."User1.Text",
                              "User2.Feedback" := "Drive_1_Auto",
                              "User2.Text" := "PLCMemory".OutputUserText.Axis1."User2.Text",
                              "User3.Feedback" := "Drive_1_RefRun",
                              "User3.Text" := "PLCMemory".OutputUserText.Axis1."User3.Text",
                              User_Text_Output => "PLCMemory".OutputUserText.Axis1.CurrentUserText);
   END_IF;
END_REGION

REGION Network 2: HMI_Start_Band_Rev
   RUNG wire#powerrail
      Contact( "HMI_Start_Band_Rev" )
      Contact( "HMI_Start_Band_Safety" )
      Coil( "Drive 1 REV]" )
   END_RUNG
   // the same network as SCL:
   "Drive 1 REV]" := "HMI_Start_Band_Rev" AND "HMI_Start_Band_Safety";
END_REGION

REGION Network 3: Drive 1 Speed 2
   RUNG wire#powerrail
      Contact( "Drive_1_Auto" )
      wire#w1
      Contact( "Drive 1 RUN FWD" )
      Coil( "Drive 1 Speed 1" )
   END_RUNG
   RUNG wire#powerrail
      Contact( "Drive_1_Manual" )
   END_RUNG wire#w1
   // the same network as SCL:
   "Drive 1 Speed 1" := ("Drive_1_Auto" OR "Drive_1_Manual") AND "Drive 1 RUN FWD";
END_REGION

REGION Network 4: Drive 2 - Control
   RUNG wire#powerrail
      "Ouput_Function_1_Drive2"("Stop Contact" := "Stop_drive_2", "Manual Command" := "Drive_2_Manual", "Auto Command" := "Drive_2_Auto", "Option Command" :=, "Disable Command" := "TurnOffDrive2", "Disable Command 2" := "PLCMemory".Disable_Modules.Disable_Trilgoten, StartScreenManual :=, Safety_StartScreenManual :=, "Ouput Signal" => "Drive 2 RUN FWD")
      "FB_OutputUsers_Axis2"("User1.Feedback" := "Drive_2_Manual", "User1.Text" := "PLCMemory".OutputUserText.Axis2."User1.Text", "User2.Feedback" := "Drive_2_Auto", "User2.Text" := "PLCMemory".OutputUserText.Axis2."User2.Text", "User3.Feedback" :=, "User3.Text" :=, "User4.Feedback" :=, "User4.Text" :=, User_Text_Output => "PLCMemory".OutputUserText.Axis2.CurrentUserText)
   END_RUNG
   // the same network as SCL:
   "Ouput_Function_1_Drive2"("Stop Contact" := "Stop_drive_2",   // "Ouput_Function_1"
                           "Manual Command" := "Drive_2_Manual",
                           "Auto Command" := "Drive_2_Auto",
                           "Disable Command" := "TurnOffDrive2",
                           "Disable Command 2" := "PLCMemory".Disable_Modules.Disable_Trilgoten,
                           "Ouput Signal" => "Drive 2 RUN FWD",
                           ENO => #_w1);
   IF #_w1 THEN
       "FB_OutputUsers_Axis2"("User1.Feedback" := "Drive_2_Manual",   // "FB_OutputUsers"
                              "User1.Text" := "PLCMemory".OutputUserText.Axis2."User1.Text",
                              "User2.Feedback" := "Drive_2_Auto",
                              "User2.Text" := "PLCMemory".OutputUserText.Axis2."User2.Text",
                              User_Text_Output => "PLCMemory".OutputUserText.Axis2.CurrentUserText);
   END_IF;
END_REGION

REGION Network 5: Drive 3 - Control (Currently controlled by Servo Drive Manager!)
   RUNG wire#powerrail
      "Ouput_Function_1_Drive3"("Stop Contact" := "Stop_drive_3", "Manual Command" := "Drive_3_Manual", "Auto Command" := "Drive_3_Auto", "Option Command" :=, "Disable Command" :=, "Disable Command 2" :=, StartScreenManual :=, Safety_StartScreenManual :=, "Ouput Signal" =>)
   END_RUNG
   // the same network as SCL:
   "Ouput_Function_1_Drive3"("Stop Contact" := "Stop_drive_3",   // "Ouput_Function_1"
                           "Manual Command" := "Drive_3_Manual",
                           "Auto Command" := "Drive_3_Auto");
END_REGION

REGION Network 6: Drive 4 - Control
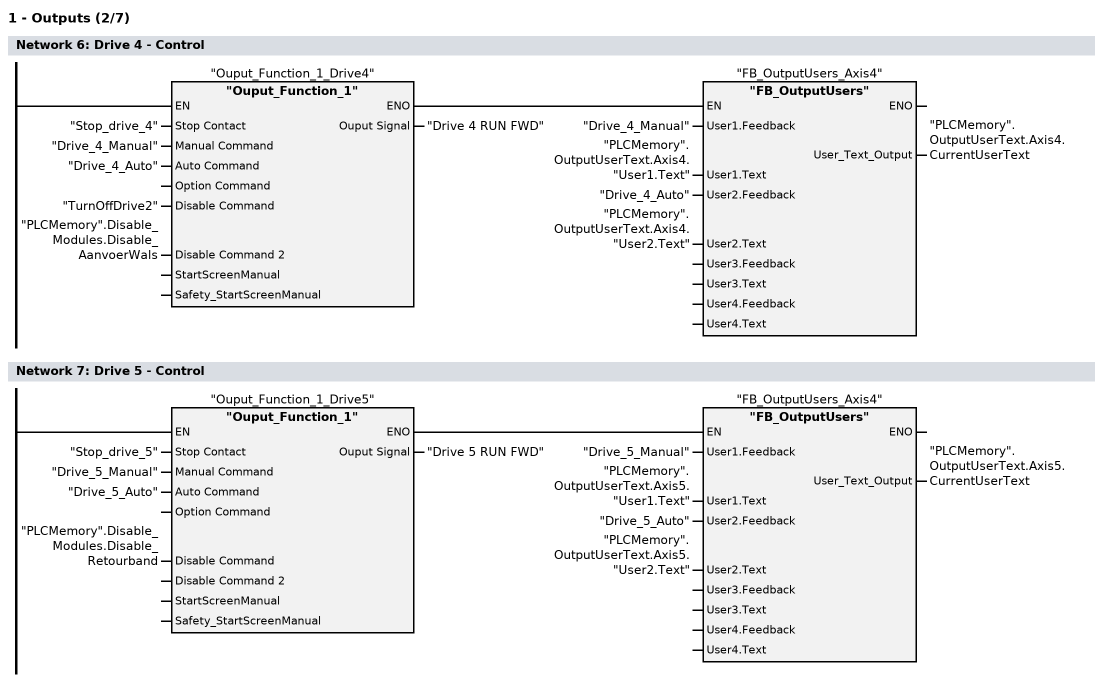
   RUNG wire#powerrail
      "Ouput_Function_1_Drive4"("Stop Contact" := "Stop_drive_4", "Manual Command" := "Drive_4_Manual", "Auto Command" := "Drive_4_Auto", "Option Command" :=, "Disable Command" := "TurnOffDrive2", "Disable Command 2" := "PLCMemory".Disable_Modules.Disable_AanvoerWals, StartScreenManual :=, Safety_StartScreenManual :=, "Ouput Signal" => "Drive 4 RUN FWD")
      "FB_OutputUsers_Axis4"("User1.Feedback" := "Drive_4_Manual", "User1.Text" := "PLCMemory".OutputUserText.Axis4."User1.Text", "User2.Feedback" := "Drive_4_Auto", "User2.Text" := "PLCMemory".OutputUserText.Axis4."User2.Text", "User3.Feedback" :=, "User3.Text" :=, "User4.Feedback" :=, "User4.Text" :=, User_Text_Output => "PLCMemory".OutputUserText.Axis4.CurrentUserText)
   END_RUNG
   // the same network as SCL:
   "Ouput_Function_1_Drive4"("Stop Contact" := "Stop_drive_4",   // "Ouput_Function_1"
                           "Manual Command" := "Drive_4_Manual",
                           "Auto Command" := "Drive_4_Auto",
                           "Disable Command" := "TurnOffDrive2",
                           "Disable Command 2" := "PLCMemory".Disable_Modules.Disable_AanvoerWals,
                           "Ouput Signal" => "Drive 4 RUN FWD",
                           ENO => #_w1);
   IF #_w1 THEN
       "FB_OutputUsers_Axis4"("User1.Feedback" := "Drive_4_Manual",   // "FB_OutputUsers"
                              "User1.Text" := "PLCMemory".OutputUserText.Axis4."User1.Text",
                              "User2.Feedback" := "Drive_4_Auto",
                              "User2.Text" := "PLCMemory".OutputUserText.Axis4."User2.Text",
                              User_Text_Output => "PLCMemory".OutputUserText.Axis4.CurrentUserText);
   END_IF;
END_REGION

REGION Network 7: Drive 5 - Control
   RUNG wire#powerrail
      "Ouput_Function_1_Drive5"("Stop Contact" := "Stop_drive_5", "Manual Command" := "Drive_5_Manual", "Auto Command" := "Drive_5_Auto", "Option Command" :=, "Disable Command" := "PLCMemory".Disable_Modules.Disable_Retourband, "Disable Command 2" :=, StartScreenManual :=, Safety_StartScreenManual :=, "Ouput Signal" => "Drive 5 RUN FWD")
      "FB_OutputUsers_Axis4"("User1.Feedback" := "Drive_5_Manual", "User1.Text" := "PLCMemory".OutputUserText.Axis5."User1.Text", "User2.Feedback" := "Drive_5_Auto", "User2.Text" := "PLCMemory".OutputUserText.Axis5."User2.Text", "User3.Feedback" :=, "User3.Text" :=, "User4.Feedback" :=, "User4.Text" :=, User_Text_Output => "PLCMemory".OutputUserText.Axis5.CurrentUserText)
   END_RUNG
   // the same network as SCL:
   "Ouput_Function_1_Drive5"("Stop Contact" := "Stop_drive_5",   // "Ouput_Function_1"
                           "Manual Command" := "Drive_5_Manual",
                           "Auto Command" := "Drive_5_Auto",
                           "Disable Command" := "PLCMemory".Disable_Modules.Disable_Retourband,
                           "Ouput Signal" => "Drive 5 RUN FWD",
                           ENO => #_w1);
   IF #_w1 THEN
       "FB_OutputUsers_Axis4"("User1.Feedback" := "Drive_5_Manual",   // "FB_OutputUsers"
                              "User1.Text" := "PLCMemory".OutputUserText.Axis5."User1.Text",
                              "User2.Feedback" := "Drive_5_Auto",
                              "User2.Text" := "PLCMemory".OutputUserText.Axis5."User2.Text",
                              User_Text_Output => "PLCMemory".OutputUserText.Axis5.CurrentUserText);
   END_IF;
END_REGION

REGION Network 8: Valve 1 - Control
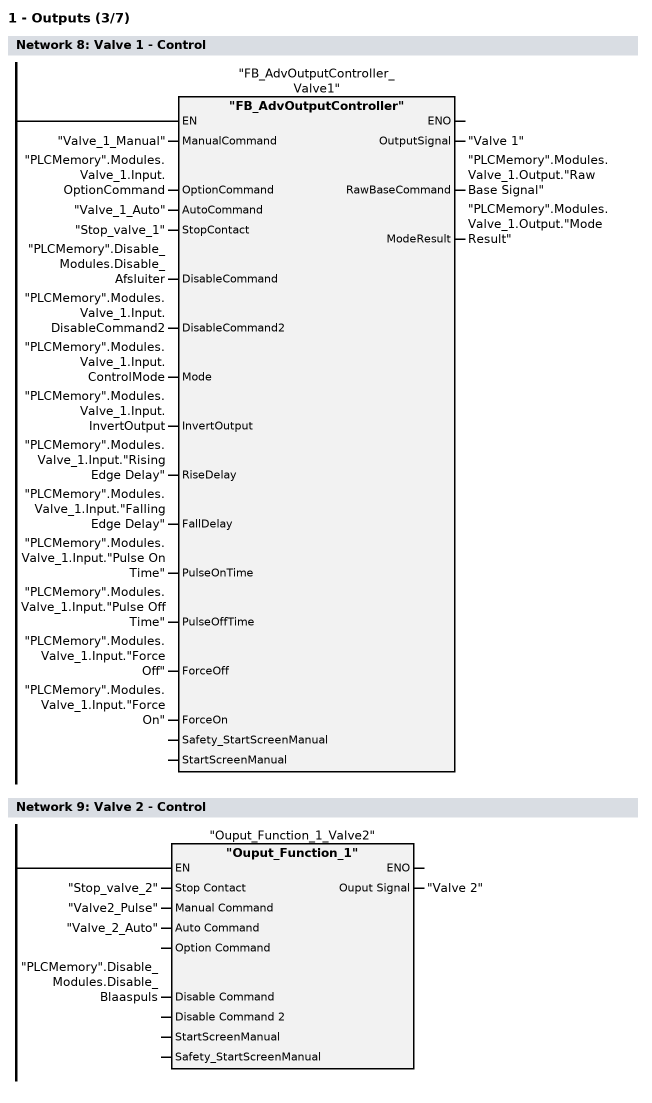
   RUNG wire#powerrail
      "FB_AdvOutputController_Valve1"(ManualCommand := "Valve_1_Manual", OptionCommand := "PLCMemory".Modules.Valve_1.Input.OptionCommand, AutoCommand := "Valve_1_Auto", StopContact := "Stop_valve_1", DisableCommand := "PLCMemory".Disable_Modules.Disable_Afsluiter, DisableCommand2 := "PLCMemory".Modules.Valve_1.Input.DisableCommand2, Mode := "PLCMemory".Modules.Valve_1.Input.ControlMode, InvertOutput := "PLCMemory".Modules.Valve_1.Input.InvertOutput, RiseDelay := "PLCMemory".Modules.Valve_1.Input."Rising Edge Delay", FallDelay := "PLCMemory".Modules.Valve_1.Input."Falling Edge Delay", PulseOnTime := "PLCMemory".Modules.Valve_1.Input."Pulse On Time", PulseOffTime := "PLCMemory".Modules.Valve_1.Input."Pulse Off Time", ForceOff := "PLCMemory".Modules.Valve_1.Input."Force Off", ForceOn := "PLCMemory".Modules.Valve_1.Input."Force On", Safety_StartScreenManual :=, StartScreenManual :=, OutputSignal => "Valve 1", RawBaseCommand => "PLCMemory".Modules.Valve_1.Output."Raw Base Signal", ModeResult => "PLCMemory".Modules.Valve_1.Output."Mode Result")
   END_RUNG
   // the same network as SCL:
   "FB_AdvOutputController_Valve1"(ManualCommand := "Valve_1_Manual",   // "FB_AdvOutputController"
                           OptionCommand := "PLCMemory".Modules.Valve_1.Input.OptionCommand,
                           AutoCommand := "Valve_1_Auto",
                           StopContact := "Stop_valve_1",
                           DisableCommand := "PLCMemory".Disable_Modules.Disable_Afsluiter,
                           DisableCommand2 := "PLCMemory".Modules.Valve_1.Input.DisableCommand2,
                           Mode := "PLCMemory".Modules.Valve_1.Input.ControlMode,
                           InvertOutput := "PLCMemory".Modules.Valve_1.Input.InvertOutput,
                           RiseDelay := "PLCMemory".Modules.Valve_1.Input."Rising Edge Delay",
                           FallDelay := "PLCMemory".Modules.Valve_1.Input."Falling Edge Delay",
                           PulseOnTime := "PLCMemory".Modules.Valve_1.Input."Pulse On Time",
                           PulseOffTime := "PLCMemory".Modules.Valve_1.Input."Pulse Off Time",
                           ForceOff := "PLCMemory".Modules.Valve_1.Input."Force Off",
                           ForceOn := "PLCMemory".Modules.Valve_1.Input."Force On",
                           OutputSignal => "Valve 1",
                           RawBaseCommand => "PLCMemory".Modules.Valve_1.Output."Raw Base Signal",
                           ModeResult => "PLCMemory".Modules.Valve_1.Output."Mode Result");
END_REGION

REGION Network 9: Valve 2 - Control
   RUNG wire#powerrail
      "Ouput_Function_1_Valve2"("Stop Contact" := "Stop_valve_2", "Manual Command" := "Valve2_Pulse", "Auto Command" := "Valve_2_Auto", "Option Command" :=, "Disable Command" := "PLCMemory".Disable_Modules.Disable_Blaaspuls, "Disable Command 2" :=, StartScreenManual :=, Safety_StartScreenManual :=, "Ouput Signal" => "Valve 2")
   END_RUNG
   // the same network as SCL:
   "Ouput_Function_1_Valve2"("Stop Contact" := "Stop_valve_2",   // "Ouput_Function_1"
                           "Manual Command" := "Valve2_Pulse",
                           "Auto Command" := "Valve_2_Auto",
                           "Disable Command" := "PLCMemory".Disable_Modules.Disable_Blaaspuls,
                           "Ouput Signal" => "Valve 2");
END_REGION

REGION Network 10: Valve 3 - Control
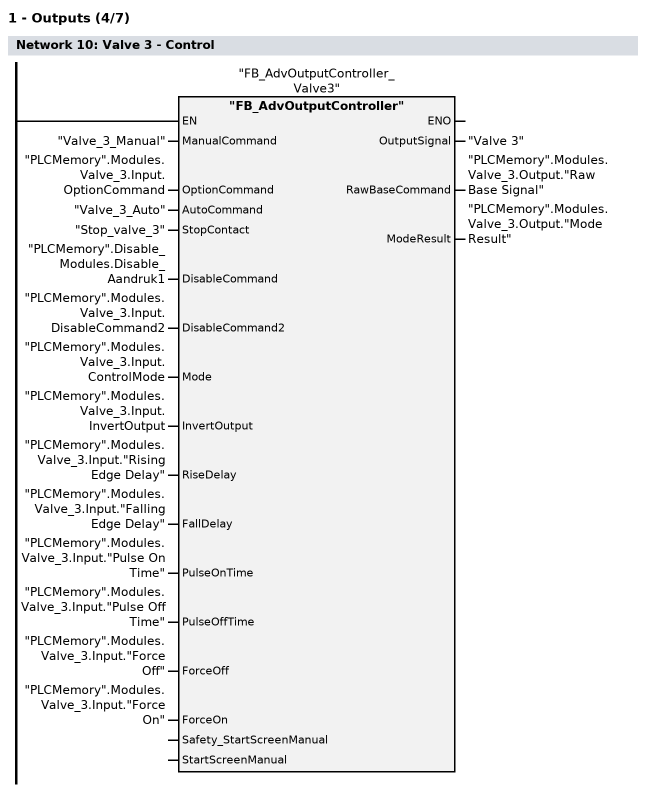
   RUNG wire#powerrail
      "FB_AdvOutputController_Valve3"(ManualCommand := "Valve_3_Manual", OptionCommand := "PLCMemory".Modules.Valve_3.Input.OptionCommand, AutoCommand := "Valve_3_Auto", StopContact := "Stop_valve_3", DisableCommand := "PLCMemory".Disable_Modules.Disable_Aandruk1, DisableCommand2 := "PLCMemory".Modules.Valve_3.Input.DisableCommand2, Mode := "PLCMemory".Modules.Valve_3.Input.ControlMode, InvertOutput := "PLCMemory".Modules.Valve_3.Input.InvertOutput, RiseDelay := "PLCMemory".Modules.Valve_3.Input."Rising Edge Delay", FallDelay := "PLCMemory".Modules.Valve_3.Input."Falling Edge Delay", PulseOnTime := "PLCMemory".Modules.Valve_3.Input."Pulse On Time", PulseOffTime := "PLCMemory".Modules.Valve_3.Input."Pulse Off Time", ForceOff := "PLCMemory".Modules.Valve_3.Input."Force Off", ForceOn := "PLCMemory".Modules.Valve_3.Input."Force On", Safety_StartScreenManual :=, StartScreenManual :=, OutputSignal => "Valve 3", RawBaseCommand => "PLCMemory".Modules.Valve_3.Output."Raw Base Signal", ModeResult => "PLCMemory".Modules.Valve_3.Output."Mode Result")
   END_RUNG
   // the same network as SCL:
   "FB_AdvOutputController_Valve3"(ManualCommand := "Valve_3_Manual",   // "FB_AdvOutputController"
                           OptionCommand := "PLCMemory".Modules.Valve_3.Input.OptionCommand,
                           AutoCommand := "Valve_3_Auto",
                           StopContact := "Stop_valve_3",
                           DisableCommand := "PLCMemory".Disable_Modules.Disable_Aandruk1,
                           DisableCommand2 := "PLCMemory".Modules.Valve_3.Input.DisableCommand2,
                           Mode := "PLCMemory".Modules.Valve_3.Input.ControlMode,
                           InvertOutput := "PLCMemory".Modules.Valve_3.Input.InvertOutput,
                           RiseDelay := "PLCMemory".Modules.Valve_3.Input."Rising Edge Delay",
                           FallDelay := "PLCMemory".Modules.Valve_3.Input."Falling Edge Delay",
                           PulseOnTime := "PLCMemory".Modules.Valve_3.Input."Pulse On Time",
                           PulseOffTime := "PLCMemory".Modules.Valve_3.Input."Pulse Off Time",
                           ForceOff := "PLCMemory".Modules.Valve_3.Input."Force Off",
                           ForceOn := "PLCMemory".Modules.Valve_3.Input."Force On",
                           OutputSignal => "Valve 3",
                           RawBaseCommand => "PLCMemory".Modules.Valve_3.Output."Raw Base Signal",
                           ModeResult => "PLCMemory".Modules.Valve_3.Output."Mode Result");
END_REGION

REGION Network 11: Valve 4 - Control
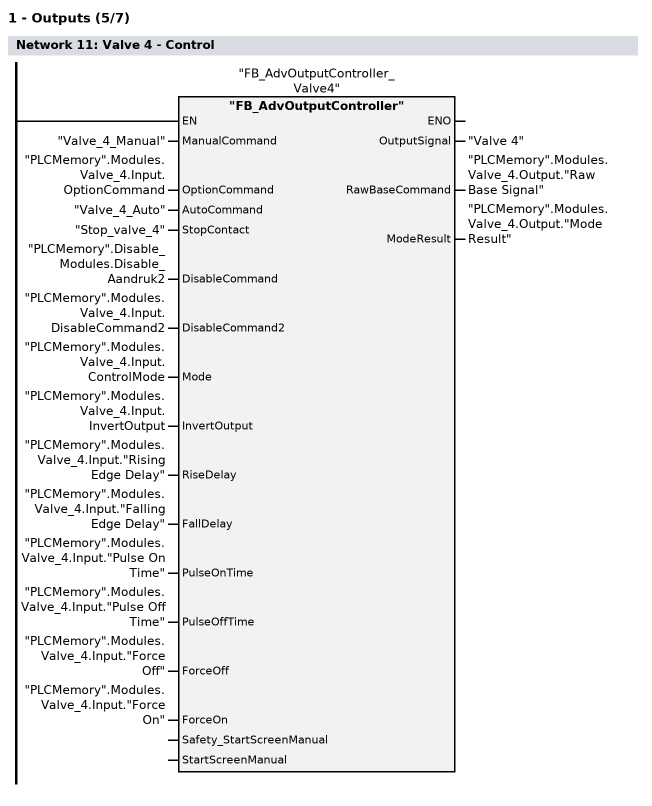
   RUNG wire#powerrail
      "FB_AdvOutputController_Valve4"(ManualCommand := "Valve_4_Manual", OptionCommand := "PLCMemory".Modules.Valve_4.Input.OptionCommand, AutoCommand := "Valve_4_Auto", StopContact := "Stop_valve_4", DisableCommand := "PLCMemory".Disable_Modules.Disable_Aandruk2, DisableCommand2 := "PLCMemory".Modules.Valve_4.Input.DisableCommand2, Mode := "PLCMemory".Modules.Valve_4.Input.ControlMode, InvertOutput := "PLCMemory".Modules.Valve_4.Input.InvertOutput, RiseDelay := "PLCMemory".Modules.Valve_4.Input."Rising Edge Delay", FallDelay := "PLCMemory".Modules.Valve_4.Input."Falling Edge Delay", PulseOnTime := "PLCMemory".Modules.Valve_4.Input."Pulse On Time", PulseOffTime := "PLCMemory".Modules.Valve_4.Input."Pulse Off Time", ForceOff := "PLCMemory".Modules.Valve_4.Input."Force Off", ForceOn := "PLCMemory".Modules.Valve_4.Input."Force On", Safety_StartScreenManual :=, StartScreenManual :=, OutputSignal => "Valve 4", RawBaseCommand => "PLCMemory".Modules.Valve_4.Output."Raw Base Signal", ModeResult => "PLCMemory".Modules.Valve_4.Output."Mode Result")
   END_RUNG
   // the same network as SCL:
   "FB_AdvOutputController_Valve4"(ManualCommand := "Valve_4_Manual",   // "FB_AdvOutputController"
                           OptionCommand := "PLCMemory".Modules.Valve_4.Input.OptionCommand,
                           AutoCommand := "Valve_4_Auto",
                           StopContact := "Stop_valve_4",
                           DisableCommand := "PLCMemory".Disable_Modules.Disable_Aandruk2,
                           DisableCommand2 := "PLCMemory".Modules.Valve_4.Input.DisableCommand2,
                           Mode := "PLCMemory".Modules.Valve_4.Input.ControlMode,
                           InvertOutput := "PLCMemory".Modules.Valve_4.Input.InvertOutput,
                           RiseDelay := "PLCMemory".Modules.Valve_4.Input."Rising Edge Delay",
                           FallDelay := "PLCMemory".Modules.Valve_4.Input."Falling Edge Delay",
                           PulseOnTime := "PLCMemory".Modules.Valve_4.Input."Pulse On Time",
                           PulseOffTime := "PLCMemory".Modules.Valve_4.Input."Pulse Off Time",
                           ForceOff := "PLCMemory".Modules.Valve_4.Input."Force Off",
                           ForceOn := "PLCMemory".Modules.Valve_4.Input."Force On",
                           OutputSignal => "Valve 4",
                           RawBaseCommand => "PLCMemory".Modules.Valve_4.Output."Raw Base Signal",
                           ModeResult => "PLCMemory".Modules.Valve_4.Output."Mode Result");
END_REGION

REGION Network 12: Valve 5 - Control
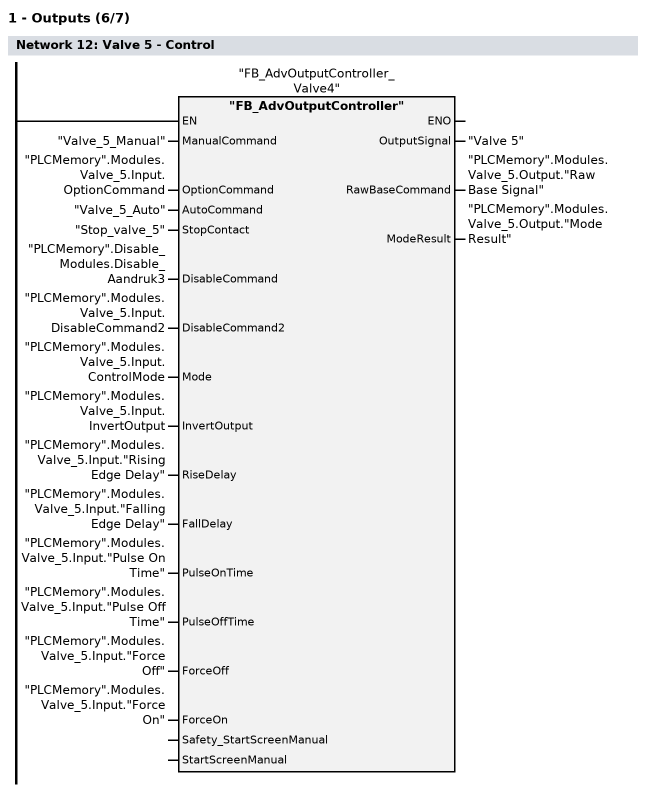
   RUNG wire#powerrail
      "FB_AdvOutputController_Valve4"(ManualCommand := "Valve_5_Manual", OptionCommand := "PLCMemory".Modules.Valve_5.Input.OptionCommand, AutoCommand := "Valve_5_Auto", StopContact := "Stop_valve_5", DisableCommand := "PLCMemory".Disable_Modules.Disable_Aandruk3, DisableCommand2 := "PLCMemory".Modules.Valve_5.Input.DisableCommand2, Mode := "PLCMemory".Modules.Valve_5.Input.ControlMode, InvertOutput := "PLCMemory".Modules.Valve_5.Input.InvertOutput, RiseDelay := "PLCMemory".Modules.Valve_5.Input."Rising Edge Delay", FallDelay := "PLCMemory".Modules.Valve_5.Input."Falling Edge Delay", PulseOnTime := "PLCMemory".Modules.Valve_5.Input."Pulse On Time", PulseOffTime := "PLCMemory".Modules.Valve_5.Input."Pulse Off Time", ForceOff := "PLCMemory".Modules.Valve_5.Input."Force Off", ForceOn := "PLCMemory".Modules.Valve_5.Input."Force On", Safety_StartScreenManual :=, StartScreenManual :=, OutputSignal => "Valve 5", RawBaseCommand => "PLCMemory".Modules.Valve_5.Output."Raw Base Signal", ModeResult => "PLCMemory".Modules.Valve_5.Output."Mode Result")
   END_RUNG
   // the same network as SCL:
   "FB_AdvOutputController_Valve4"(ManualCommand := "Valve_5_Manual",   // "FB_AdvOutputController"
                           OptionCommand := "PLCMemory".Modules.Valve_5.Input.OptionCommand,
                           AutoCommand := "Valve_5_Auto",
                           StopContact := "Stop_valve_5",
                           DisableCommand := "PLCMemory".Disable_Modules.Disable_Aandruk3,
                           DisableCommand2 := "PLCMemory".Modules.Valve_5.Input.DisableCommand2,
                           Mode := "PLCMemory".Modules.Valve_5.Input.ControlMode,
                           InvertOutput := "PLCMemory".Modules.Valve_5.Input.InvertOutput,
                           RiseDelay := "PLCMemory".Modules.Valve_5.Input."Rising Edge Delay",
                           FallDelay := "PLCMemory".Modules.Valve_5.Input."Falling Edge Delay",
                           PulseOnTime := "PLCMemory".Modules.Valve_5.Input."Pulse On Time",
                           PulseOffTime := "PLCMemory".Modules.Valve_5.Input."Pulse Off Time",
                           ForceOff := "PLCMemory".Modules.Valve_5.Input."Force Off",
                           ForceOn := "PLCMemory".Modules.Valve_5.Input."Force On",
                           OutputSignal => "Valve 5",
                           RawBaseCommand => "PLCMemory".Modules.Valve_5.Output."Raw Base Signal",
                           ModeResult => "PLCMemory".Modules.Valve_5.Output."Mode Result");
END_REGION

REGION Network 13: Valve 6 - Control
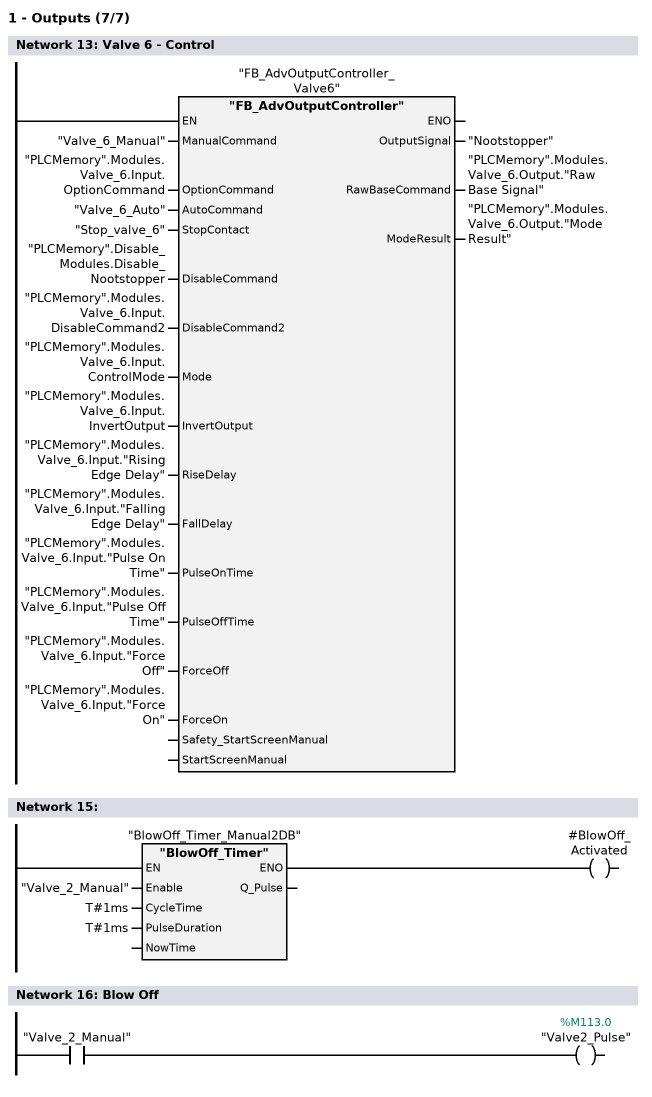
   RUNG wire#powerrail
      "FB_AdvOutputController_Valve6"(ManualCommand := "Valve_6_Manual", OptionCommand := "PLCMemory".Modules.Valve_6.Input.OptionCommand, AutoCommand := "Valve_6_Auto", StopContact := "Stop_valve_6", DisableCommand := "PLCMemory".Disable_Modules.Disable_Nootstopper, DisableCommand2 := "PLCMemory".Modules.Valve_6.Input.DisableCommand2, Mode := "PLCMemory".Modules.Valve_6.Input.ControlMode, InvertOutput := "PLCMemory".Modules.Valve_6.Input.InvertOutput, RiseDelay := "PLCMemory".Modules.Valve_6.Input."Rising Edge Delay", FallDelay := "PLCMemory".Modules.Valve_6.Input."Falling Edge Delay", PulseOnTime := "PLCMemory".Modules.Valve_6.Input."Pulse On Time", PulseOffTime := "PLCMemory".Modules.Valve_6.Input."Pulse Off Time", ForceOff := "PLCMemory".Modules.Valve_6.Input."Force Off", ForceOn := "PLCMemory".Modules.Valve_6.Input."Force On", Safety_StartScreenManual :=, StartScreenManual :=, OutputSignal => "Nootstopper", RawBaseCommand => "PLCMemory".Modules.Valve_6.Output."Raw Base Signal", ModeResult => "PLCMemory".Modules.Valve_6.Output."Mode Result")
   END_RUNG
   // the same network as SCL:
   "FB_AdvOutputController_Valve6"(ManualCommand := "Valve_6_Manual",   // "FB_AdvOutputController"
                           OptionCommand := "PLCMemory".Modules.Valve_6.Input.OptionCommand,
                           AutoCommand := "Valve_6_Auto",
                           StopContact := "Stop_valve_6",
                           DisableCommand := "PLCMemory".Disable_Modules.Disable_Nootstopper,
                           DisableCommand2 := "PLCMemory".Modules.Valve_6.Input.DisableCommand2,
                           Mode := "PLCMemory".Modules.Valve_6.Input.ControlMode,
                           InvertOutput := "PLCMemory".Modules.Valve_6.Input.InvertOutput,
                           RiseDelay := "PLCMemory".Modules.Valve_6.Input."Rising Edge Delay",
                           FallDelay := "PLCMemory".Modules.Valve_6.Input."Falling Edge Delay",
                           PulseOnTime := "PLCMemory".Modules.Valve_6.Input."Pulse On Time",
                           PulseOffTime := "PLCMemory".Modules.Valve_6.Input."Pulse Off Time",
                           ForceOff := "PLCMemory".Modules.Valve_6.Input."Force Off",
                           ForceOn := "PLCMemory".Modules.Valve_6.Input."Force On",
                           OutputSignal => "Nootstopper",
                           RawBaseCommand => "PLCMemory".Modules.Valve_6.Output."Raw Base Signal",
                           ModeResult => "PLCMemory".Modules.Valve_6.Output."Mode Result");
END_REGION

REGION Network 14: Blow Off Manual
END_REGION

REGION Network 15
   RUNG wire#powerrail
      "BlowOff_Timer_Manual2DB"(Enable := "Valve_2_Manual", CycleTime := T#1ms, PulseDuration := T#1ms, NowTime :=, Q_Pulse =>)
      Coil( #BlowOff_Activated )
   END_RUNG
   // the same network as SCL:
   "BlowOff_Timer_Manual2DB"(Enable := "Valve_2_Manual",   // "BlowOff_Timer"
                           CycleTime := T#1ms,
                           PulseDuration := T#1ms,
                           ENO => #_w1);
   #BlowOff_Activated := #_w1;
END_REGION

REGION Network 16: Blow Off
   RUNG wire#powerrail
      Contact( "Valve_2_Manual" )
      Coil( "Valve2_Pulse" )
   END_RUNG
   // the same network as SCL:
   "Valve2_Pulse" := "Valve_2_Manual";
END_REGION
END_FUNCTION

FUNCTION_BLOCK "Ouput_Function_1"   // FB8, FBD
TITLE = Ouput Controller Function Block
VERSION : 0.1
// stored: AutoNumber true, IsIECCheckEnabled false, UDAEnableTagReadback false
   VAR_INPUT
      "Stop Contact" : Bool;
      "Manual Command" : Bool;
      "Auto Command" : Bool;
      "Option Command" : Bool;
      "Disable Command" : Bool;
      "Disable Command 2" : Bool;
      StartScreenManual : Bool;
      Safety_StartScreenManual : Bool;
   END_VAR
   VAR_OUTPUT
      "Ouput Signal" : Bool;
   END_VAR
BEGIN

REGION Network 1: Ouput Controller
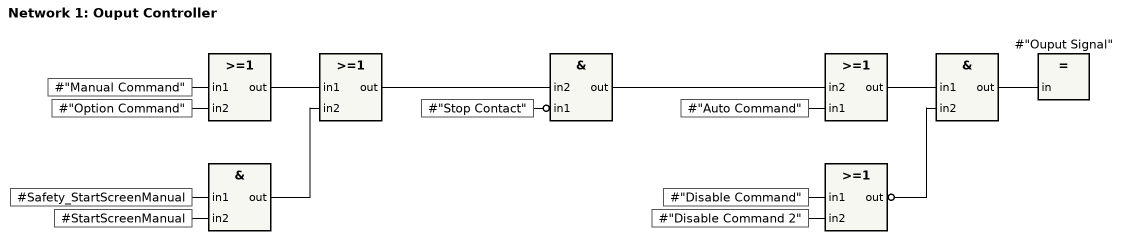
   #"Ouput Signal" := (((#"Manual Command" OR #"Option Command" OR (#Safety_StartScreenManual AND #StartScreenManual)) AND NOT #"Stop Contact") OR #"Auto Command") AND NOT (#"Disable Command" OR #"Disable Command 2");
END_REGION
END_FUNCTION_BLOCK

FUNCTION "6 - Storingsmelding" : Void   // FC8, LAD
TITLE = Warnings
VERSION : 0.1
// This program block is for audible & visual warnings.
// stored: AutoNumber true, IsIECCheckEnabled false, UDAEnableTagReadback false
   VAR_TEMP
      "Wals Sensor Controlled" : Bool;
      "Infeed Sensor Controlled" : Bool;
      EnoughProductsOnInfeed : Bool;
      NotEnoughProductsOnInfeed : Bool;
      Warning_NotEnoughProducts : Bool;
      TurnOffDrives : Bool;
   END_VAR
   VAR CONSTANT
      "Sensor 2 (option)" : Bool := TRUE;
   END_VAR
   VAR_TEMP   // added for the SCL form of the ladder/FBD networks
      _w1 : Bool;
   END_VAR
BEGIN

REGION Network 1: +MC-21K6:5 - Bel Storing
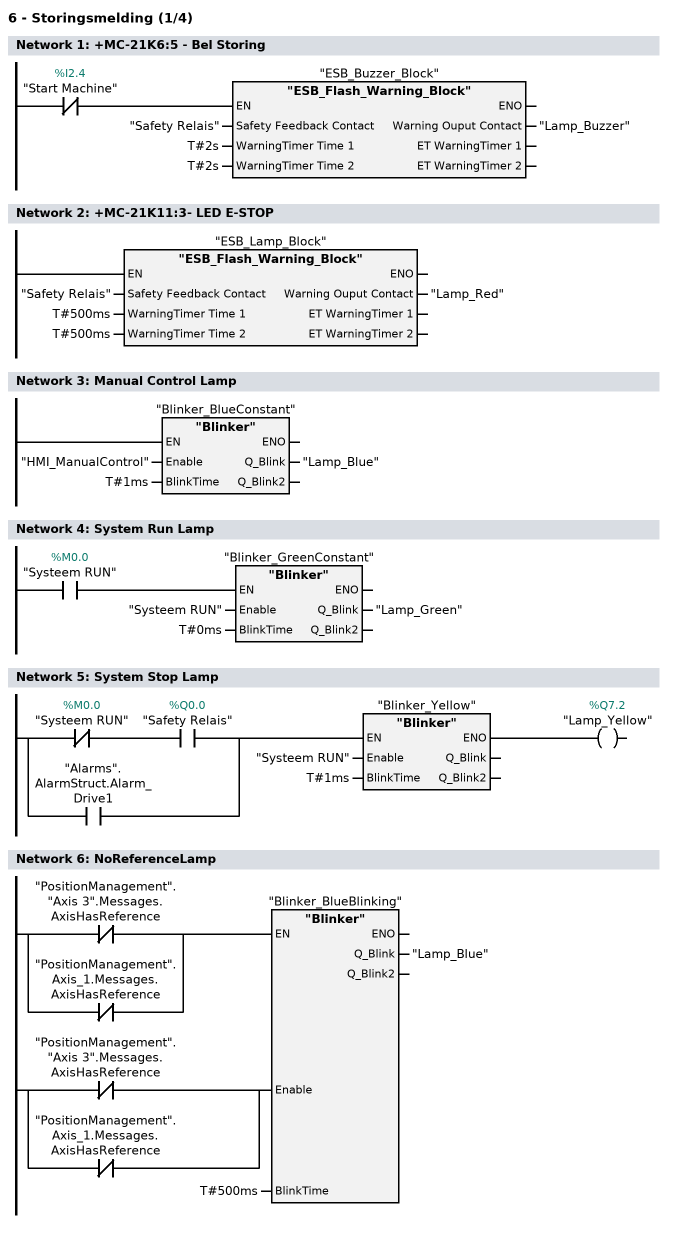
   RUNG wire#powerrail
      I_Contact( "Start Machine" )
      "ESB_Buzzer_Block"("Safety Feedback Contact" := "Safety Relais", "WarningTimer Time 1" := T#2s, "WarningTimer Time 2" := T#2s, "Warning Ouput Contact" => "Lamp_Buzzer", "ET WarningTimer 1" =>, "ET WarningTimer 2" =>)
   END_RUNG
   // the same network as SCL:
   IF NOT "Start Machine" THEN
       "ESB_Buzzer_Block"("Safety Feedback Contact" := "Safety Relais",   // "ESB_Flash_Warning_Block"
                          "WarningTimer Time 1" := T#2s,
                          "WarningTimer Time 2" := T#2s,
                          "Warning Ouput Contact" => "Lamp_Buzzer");
   END_IF;
END_REGION

REGION Network 2: +MC-21K11:3- LED E-STOP
   RUNG wire#powerrail
      "ESB_Lamp_Block"("Safety Feedback Contact" := "Safety Relais", "WarningTimer Time 1" := T#500ms, "WarningTimer Time 2" := T#500ms, "Warning Ouput Contact" => "Lamp_Red", "ET WarningTimer 1" =>, "ET WarningTimer 2" =>)
   END_RUNG
   // the same network as SCL:
   "ESB_Lamp_Block"("Safety Feedback Contact" := "Safety Relais",   // "ESB_Flash_Warning_Block"
                    "WarningTimer Time 1" := T#500ms,
                    "WarningTimer Time 2" := T#500ms,
                    "Warning Ouput Contact" => "Lamp_Red");
END_REGION

REGION Network 3: Manual Control Lamp
   RUNG wire#powerrail
      "Blinker_BlueConstant"(Enable := "HMI_ManualControl", BlinkTime := T#1ms, Q_Blink => "Lamp_Blue", Q_Blink2 =>)
   END_RUNG
   // the same network as SCL:
   "Blinker_BlueConstant"(Enable := "HMI_ManualControl", BlinkTime := T#1ms, Q_Blink => "Lamp_Blue");   // "Blinker"
END_REGION

REGION Network 4: System Run Lamp
   RUNG wire#powerrail
      Contact( "Systeem RUN" )
      "Blinker_GreenConstant"(Enable := "Systeem RUN", BlinkTime := T#0ms, Q_Blink => "Lamp_Green", Q_Blink2 =>)
   END_RUNG
   // the same network as SCL:
   IF "Systeem RUN" THEN
       "Blinker_GreenConstant"(Enable := "Systeem RUN", BlinkTime := T#0ms, Q_Blink => "Lamp_Green");   // "Blinker"
   END_IF;
END_REGION

REGION Network 5: System Stop Lamp
   RUNG wire#powerrail
      I_Contact( "Systeem RUN" )
      Contact( "Safety Relais" )
      wire#w1
      "Blinker_Yellow"(Enable := "Systeem RUN", BlinkTime := T#1ms, Q_Blink =>, Q_Blink2 =>)
      Coil( "Lamp_Yellow" )
   END_RUNG
   RUNG wire#powerrail
      Contact( "Alarms".AlarmStruct.Alarm_Drive1 )
   END_RUNG wire#w1
   // the same network as SCL:
   "Blinker_Yellow"(EN := (NOT "Systeem RUN" AND "Safety Relais") OR "Alarms".AlarmStruct.Alarm_Drive1,   // "Blinker"
                    Enable := "Systeem RUN",
                    BlinkTime := T#1ms,
                    ENO => #_w1);
   "Lamp_Yellow" := #_w1;
END_REGION

REGION Network 6: NoReferenceLamp
   RUNG wire#powerrail
      I_Contact( "PositionManagement"."Axis 3".Messages.AxisHasReference )
      wire#w1
      "Blinker_BlueBlinking"(Enable := wire#w2, BlinkTime := T#500ms, Q_Blink => "Lamp_Blue", Q_Blink2 =>)
   END_RUNG
   RUNG wire#powerrail
      I_Contact( "PositionManagement".Axis_1.Messages.AxisHasReference )
   END_RUNG wire#w1
   RUNG wire#powerrail
      I_Contact( "PositionManagement"."Axis 3".Messages.AxisHasReference )
   END_RUNG wire#w2
   RUNG wire#powerrail
      I_Contact( "PositionManagement".Axis_1.Messages.AxisHasReference )
   END_RUNG wire#w2
   // the same network as SCL:
   IF NOT "PositionManagement"."Axis 3".Messages.AxisHasReference OR NOT "PositionManagement".Axis_1.Messages.AxisHasReference THEN
       "Blinker_BlueBlinking"(Enable := NOT "PositionManagement"."Axis 3".Messages.AxisHasReference OR NOT "PositionManagement".Axis_1.Messages.AxisHasReference,   // "Blinker"
                              BlinkTime := T#500ms,
                              Q_Blink => "Lamp_Blue");
   END_IF;
END_REGION

REGION Network 7: Fill Trechter Delay Function
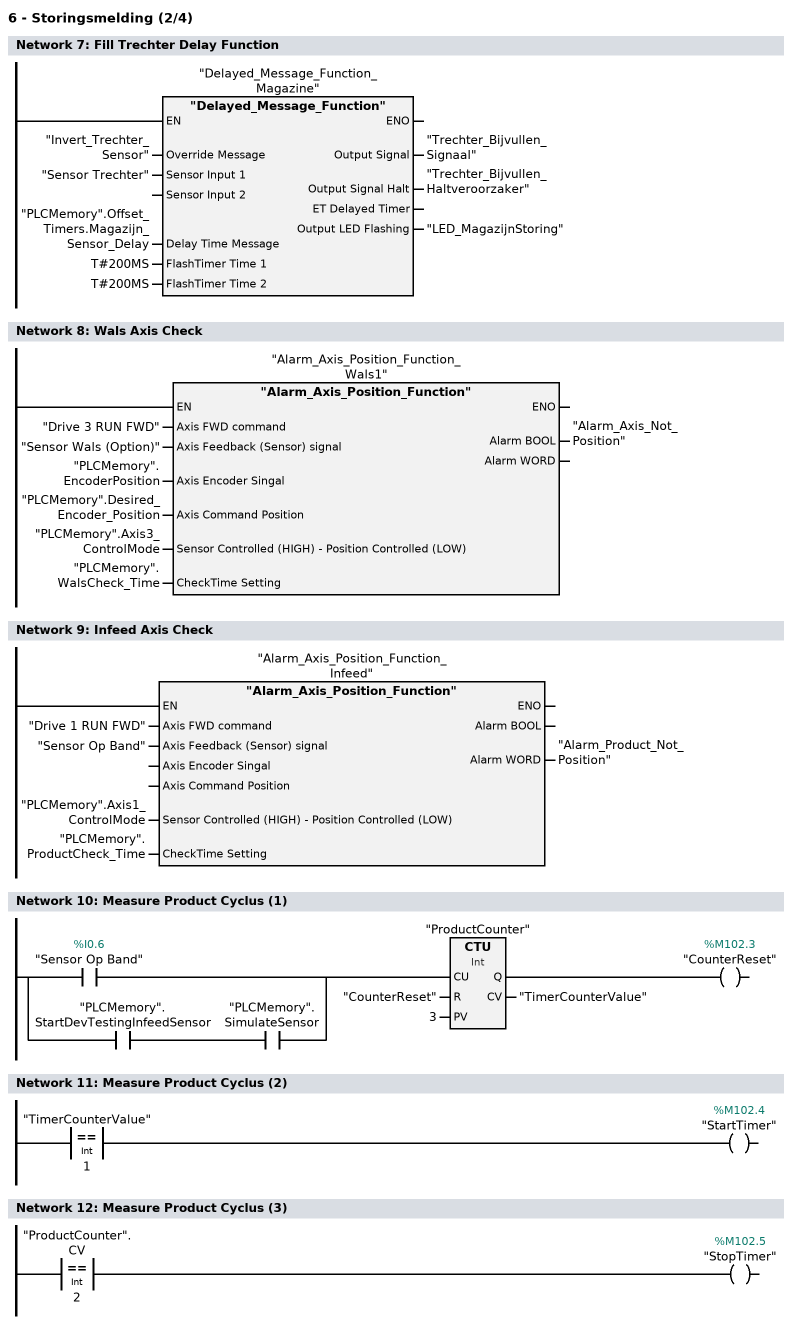
   RUNG wire#powerrail
      "Delayed_Message_Function_Magazine"("Override Message" := "Invert_Trechter_Sensor", "Sensor Input 1" := "Sensor Trechter", "Sensor Input 2" :=, "Delay Time Message" := "PLCMemory".Offset_Timers.Magazijn_Sensor_Delay, "FlashTimer Time 1" := T#200MS, "FlashTimer Time 2" := T#200MS, "Output Signal" => "Trechter_Bijvullen_Signaal", "Output Signal Halt" => "Trechter_Bijvullen_Haltveroorzaker", "ET Delayed Timer" =>, "Output LED Flashing" => "LED_MagazijnStoring")
   END_RUNG
   // the same network as SCL:
   "Delayed_Message_Function_Magazine"("Override Message" := "Invert_Trechter_Sensor",   // "Delayed_Message_Function"
                           "Sensor Input 1" := "Sensor Trechter",
                           "Delay Time Message" := "PLCMemory".Offset_Timers.Magazijn_Sensor_Delay,
                           "FlashTimer Time 1" := T#200MS,
                           "FlashTimer Time 2" := T#200MS,
                           "Output Signal" => "Trechter_Bijvullen_Signaal",
                           "Output Signal Halt" => "Trechter_Bijvullen_Haltveroorzaker",
                           "Output LED Flashing" => "LED_MagazijnStoring");
END_REGION

REGION Network 8: Wals Axis Check
   RUNG wire#powerrail
      "Alarm_Axis_Position_Function_Wals1"("Axis FWD command" := "Drive 3 RUN FWD", "Axis Feedback (Sensor) signal" := "Sensor Wals (Option)", "Axis Encoder Singal" := "PLCMemory".EncoderPosition, "Axis Command Position" := "PLCMemory".Desired_Encoder_Position, "Sensor Controlled (HIGH) - Position Controlled (LOW)" := "PLCMemory".Axis3_ControlMode, "CheckTime Setting" := "PLCMemory".WalsCheck_Time, "Alarm BOOL" => "Alarm_Axis_Not_Position", "Alarm WORD" =>)
   END_RUNG
   // the same network as SCL:
   "Alarm_Axis_Position_Function_Wals1"("Axis FWD command" := "Drive 3 RUN FWD",   // "Alarm_Axis_Position_Function"
                           "Axis Feedback (Sensor) signal" := "Sensor Wals (Option)",
                           "Axis Encoder Singal" := "PLCMemory".EncoderPosition,
                           "Axis Command Position" := "PLCMemory".Desired_Encoder_Position,
                           "Sensor Controlled (HIGH) - Position Controlled (LOW)" := "PLCMemory".Axis3_ControlMode,
                           "CheckTime Setting" := "PLCMemory".WalsCheck_Time,
                           "Alarm BOOL" => "Alarm_Axis_Not_Position");
END_REGION

REGION Network 9: Infeed Axis Check
   RUNG wire#powerrail
      "Alarm_Axis_Position_Function_Infeed"("Axis FWD command" := "Drive 1 RUN FWD", "Axis Feedback (Sensor) signal" := "Sensor Op Band", "Axis Encoder Singal" :=, "Axis Command Position" :=, "Sensor Controlled (HIGH) - Position Controlled (LOW)" := "PLCMemory".Axis1_ControlMode, "CheckTime Setting" := "PLCMemory".ProductCheck_Time, "Alarm BOOL" =>, "Alarm WORD" => "Alarm_Product_Not_Position")
   END_RUNG
   // the same network as SCL:
   "Alarm_Axis_Position_Function_Infeed"("Axis FWD command" := "Drive 1 RUN FWD",   // "Alarm_Axis_Position_Function"
                           "Axis Feedback (Sensor) signal" := "Sensor Op Band",
                           "Sensor Controlled (HIGH) - Position Controlled (LOW)" := "PLCMemory".Axis1_ControlMode,
                           "CheckTime Setting" := "PLCMemory".ProductCheck_Time,
                           "Alarm WORD" => "Alarm_Product_Not_Position");
END_REGION

REGION Network 10: Measure Product Cyclus (1)
   RUNG wire#powerrail
      Contact( "Sensor Op Band" )
      wire#w1
      { S7_Templates := "value_type := Int" } "ProductCounter".CTU(r := "CounterReset", pv := 3, cv => "TimerCounterValue")
      Coil( "CounterReset" )
   END_RUNG
   RUNG wire#powerrail
      Contact( "PLCMemory".StartDevTestingInfeedSensor )
      Contact( "PLCMemory".SimulateSensor )
   END_RUNG wire#w1
   // the same network as SCL:
   "ProductCounter".CTU(CU := "Sensor Op Band" OR ("PLCMemory".StartDevTestingInfeedSensor AND "PLCMemory".SimulateSensor),
                        R := "CounterReset",
                        PV := 3,
                        CV => "TimerCounterValue");
   "CounterReset" := "ProductCounter".Q;
END_REGION

REGION Network 11: Measure Product Cyclus (2)
   RUNG wire#powerrail
      { S7_Templates := "SrcType := Int" } EQ_Contact(in1 := "TimerCounterValue", in2 := 1)
      Coil( "StartTimer" )
   END_RUNG
   // the same network as SCL:
   "StartTimer" := "TimerCounterValue" = 1;
END_REGION

REGION Network 12: Measure Product Cyclus (3)
   RUNG wire#powerrail
      { S7_Templates := "SrcType := Int" } EQ_Contact(in1 := "ProductCounter".CV, in2 := 2)
      Coil( "StopTimer" )
   END_RUNG
   // the same network as SCL:
   "StopTimer" := "ProductCounter".CV = 2;
END_REGION

REGION Network 13: Measure Product Cyclus (4)
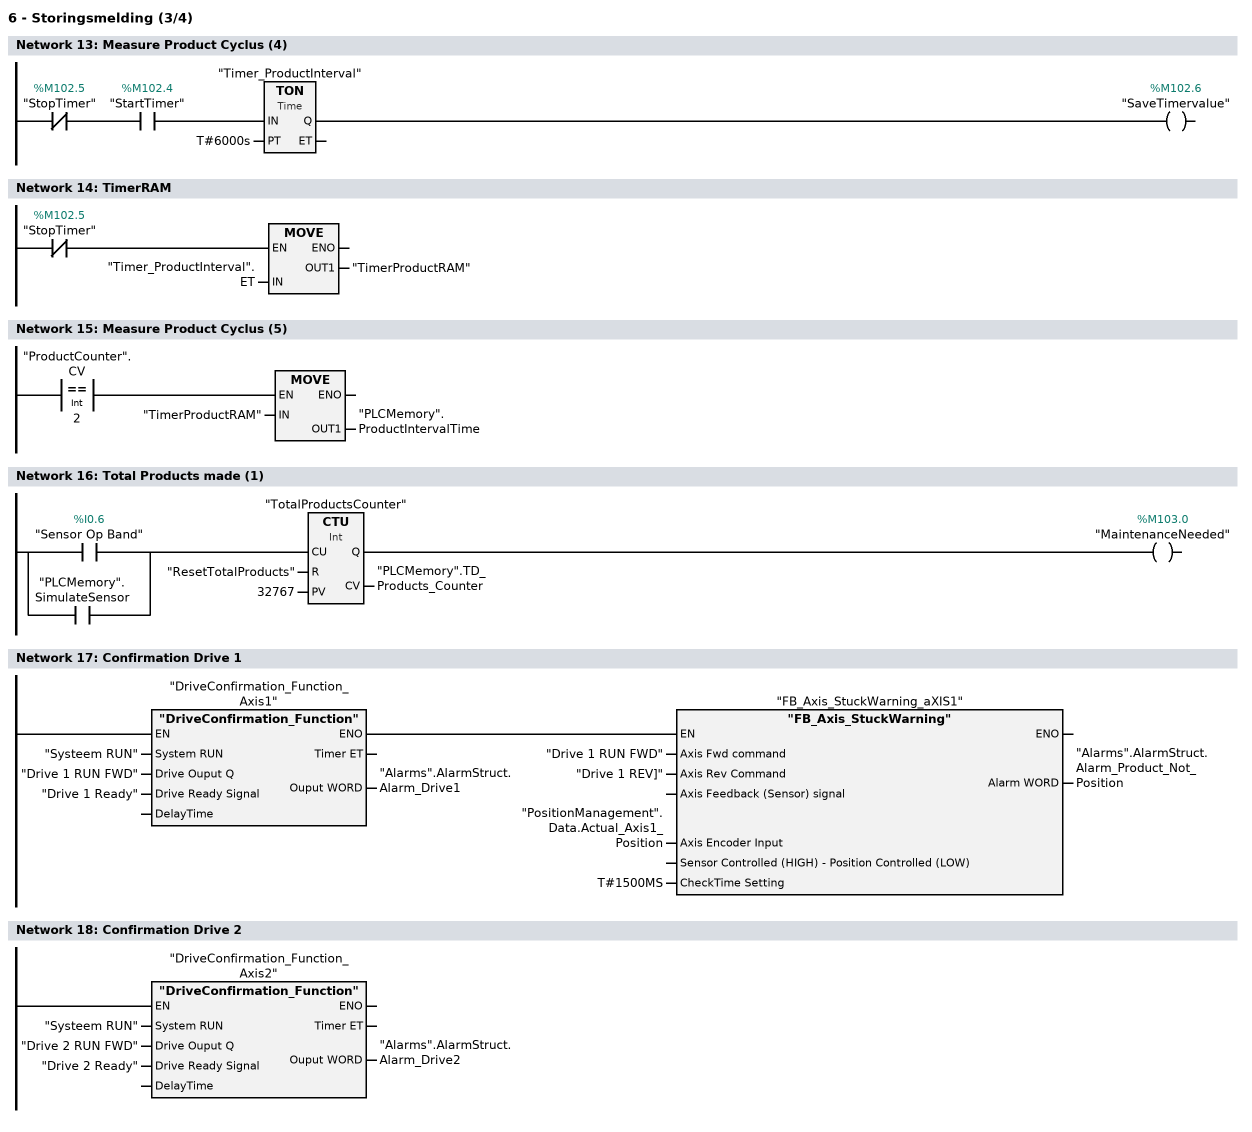
   RUNG wire#powerrail
      I_Contact( "StopTimer" )
      Contact( "StartTimer" )
      { S7_Templates := "time_type := Time" } "Timer_ProductInterval".TON(pt := T#6000s, et =>)
      Coil( "SaveTimervalue" )
   END_RUNG
   // the same network as SCL:
   "Timer_ProductInterval".TON(IN := NOT "StopTimer" AND "StartTimer", PT := T#6000s);
   "SaveTimervalue" := "Timer_ProductInterval".Q;
END_REGION

REGION Network 14: TimerRAM
   RUNG wire#powerrail
      I_Contact( "StopTimer" )
      { S7_GenerateENO := "TRUE" } Move(in := "Timer_ProductInterval".ET, out1 => "TimerProductRAM")
   END_RUNG
   // the same network as SCL:
   IF NOT "StopTimer" THEN "TimerProductRAM" := "Timer_ProductInterval".ET; END_IF;
END_REGION

REGION Network 15: Measure Product Cyclus (5)
   RUNG wire#powerrail
      { S7_Templates := "SrcType := Int" } EQ_Contact(in1 := "ProductCounter".CV, in2 := 2)
      { S7_GenerateENO := "TRUE" } Move(in := "TimerProductRAM", out1 => "PLCMemory".ProductIntervalTime)
   END_RUNG
   // the same network as SCL:
   IF "ProductCounter".CV = 2 THEN "PLCMemory".ProductIntervalTime := "TimerProductRAM"; END_IF;
END_REGION

REGION Network 16: Total Products made (1)
   RUNG wire#powerrail
      Contact( "Sensor Op Band" )
      wire#w1
      { S7_Templates := "value_type := Int" } "TotalProductsCounter".CTU(r := "ResetTotalProducts", pv := 32767, cv => "PLCMemory".TD_Products_Counter)
      Coil( "MaintenanceNeeded" )
   END_RUNG
   RUNG wire#powerrail
      Contact( "PLCMemory".SimulateSensor )
   END_RUNG wire#w1
   // the same network as SCL:
   "TotalProductsCounter".CTU(CU := "Sensor Op Band" OR "PLCMemory".SimulateSensor,
                           R := "ResetTotalProducts",
                           PV := 32767,
                           CV => "PLCMemory".TD_Products_Counter);
   "MaintenanceNeeded" := "TotalProductsCounter".Q;
END_REGION

REGION Network 17: Confirmation Drive 1
   RUNG wire#powerrail
      "DriveConfirmation_Function_Axis1"("System RUN" := "Systeem RUN", "Drive Ouput Q" := "Drive 1 RUN FWD", "Drive Ready Signal" := "Drive 1 Ready", DelayTime :=, "Timer ET" =>, "Ouput WORD" => "Alarms".AlarmStruct.Alarm_Drive1)
      "FB_Axis_StuckWarning_aXIS1"("Axis Fwd command" := "Drive 1 RUN FWD", "Axis Rev Command" := "Drive 1 REV]", "Axis Feedback (Sensor) signal" :=, "Axis Encoder Input" := "PositionManagement".Data.Actual_Axis1_Position, "Sensor Controlled (HIGH) - Position Controlled (LOW)" :=, "CheckTime Setting" := T#1500MS, "Alarm WORD" => "Alarms".AlarmStruct.Alarm_Product_Not_Position)
   END_RUNG
   // the same network as SCL:
   "DriveConfirmation_Function_Axis1"("System RUN" := "Systeem RUN",   // "DriveConfirmation_Function"
                           "Drive Ouput Q" := "Drive 1 RUN FWD",
                           "Drive Ready Signal" := "Drive 1 Ready",
                           "Ouput WORD" => "Alarms".AlarmStruct.Alarm_Drive1,
                           ENO => #_w1);
   IF #_w1 THEN
       "FB_Axis_StuckWarning_aXIS1"("Axis Fwd command" := "Drive 1 RUN FWD",   // "FB_Axis_StuckWarning"
                               "Axis Rev Command" := "Drive 1 REV]",
                               "Axis Encoder Input" := "PositionManagement".Data.Actual_Axis1_Position,
                               "CheckTime Setting" := T#1500MS,
                               "Alarm WORD" => "Alarms".AlarmStruct.Alarm_Product_Not_Position);
   END_IF;
END_REGION

REGION Network 18: Confirmation Drive 2
   RUNG wire#powerrail
      "DriveConfirmation_Function_Axis2"("System RUN" := "Systeem RUN", "Drive Ouput Q" := "Drive 2 RUN FWD", "Drive Ready Signal" := "Drive 2 Ready", DelayTime :=, "Timer ET" =>, "Ouput WORD" => "Alarms".AlarmStruct.Alarm_Drive2)
   END_RUNG
   // the same network as SCL:
   "DriveConfirmation_Function_Axis2"("System RUN" := "Systeem RUN",   // "DriveConfirmation_Function"
                           "Drive Ouput Q" := "Drive 2 RUN FWD",
                           "Drive Ready Signal" := "Drive 2 Ready",
                           "Ouput WORD" => "Alarms".AlarmStruct.Alarm_Drive2);
END_REGION

REGION Network 19: Confirmation Drive 3
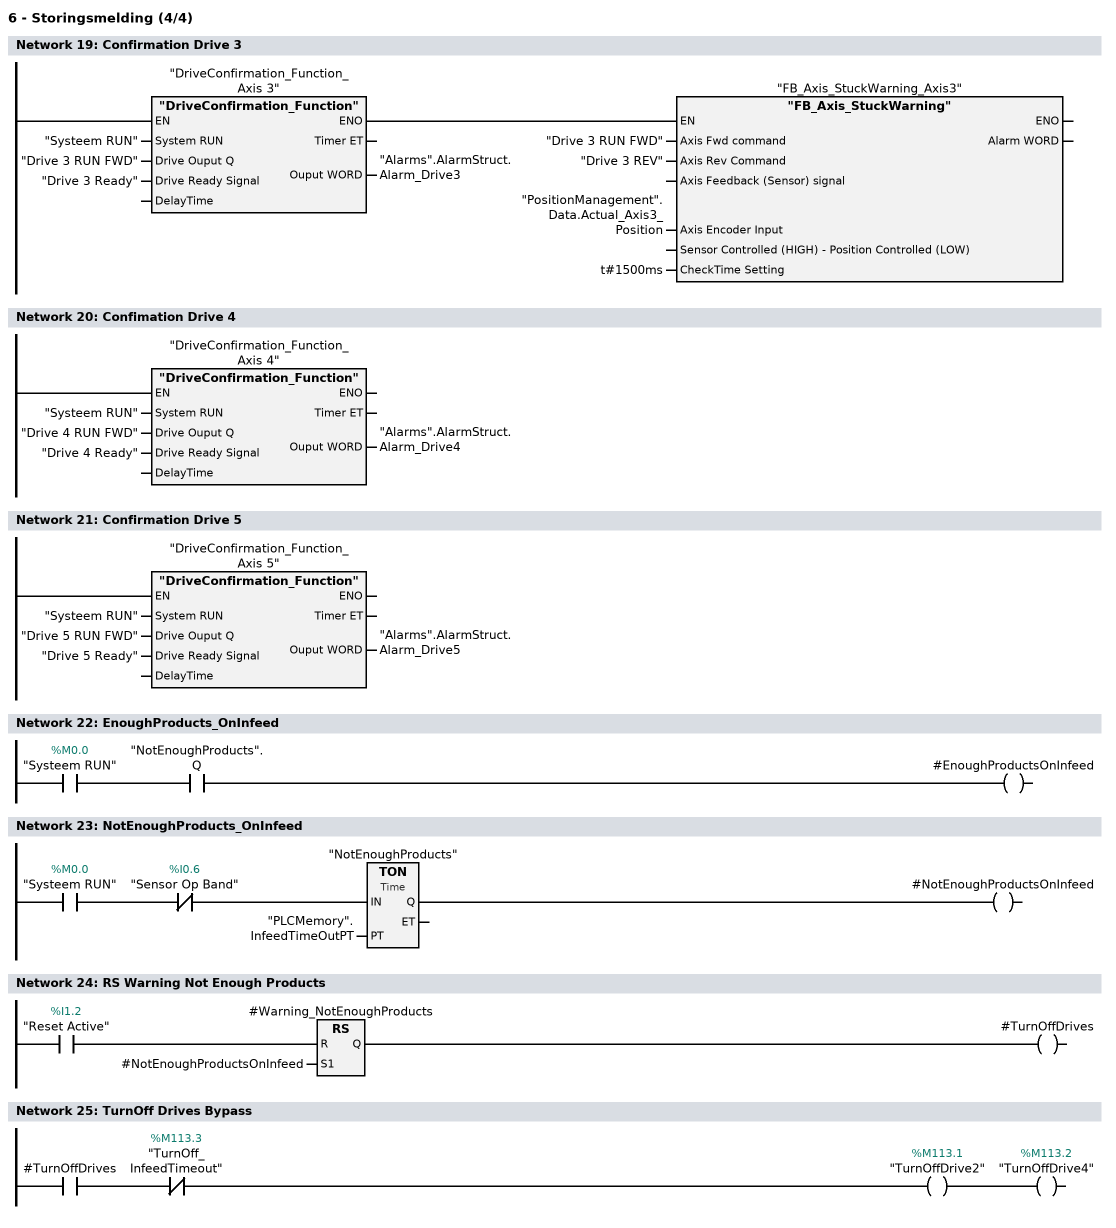
   RUNG wire#powerrail
      "DriveConfirmation_Function_Axis 3"("System RUN" := "Systeem RUN", "Drive Ouput Q" := "Drive 3 RUN FWD", "Drive Ready Signal" := "Drive 3 Ready", DelayTime :=, "Timer ET" =>, "Ouput WORD" => "Alarms".AlarmStruct.Alarm_Drive3)
      "FB_Axis_StuckWarning_Axis3"("Axis Fwd command" := "Drive 3 RUN FWD", "Axis Rev Command" := "Drive 3 REV", "Axis Feedback (Sensor) signal" :=, "Axis Encoder Input" := "PositionManagement".Data.Actual_Axis3_Position, "Sensor Controlled (HIGH) - Position Controlled (LOW)" :=, "CheckTime Setting" := t#1500ms, "Alarm WORD" =>)
   END_RUNG
   // the same network as SCL:
   "DriveConfirmation_Function_Axis 3"("System RUN" := "Systeem RUN",   // "DriveConfirmation_Function"
                           "Drive Ouput Q" := "Drive 3 RUN FWD",
                           "Drive Ready Signal" := "Drive 3 Ready",
                           "Ouput WORD" => "Alarms".AlarmStruct.Alarm_Drive3,
                           ENO => #_w1);
   IF #_w1 THEN
       "FB_Axis_StuckWarning_Axis3"("Axis Fwd command" := "Drive 3 RUN FWD",   // "FB_Axis_StuckWarning"
                               "Axis Rev Command" := "Drive 3 REV",
                               "Axis Encoder Input" := "PositionManagement".Data.Actual_Axis3_Position,
                               "CheckTime Setting" := t#1500ms);
   END_IF;
END_REGION

REGION Network 20: Confimation Drive 4
   RUNG wire#powerrail
      "DriveConfirmation_Function_Axis 4"("System RUN" := "Systeem RUN", "Drive Ouput Q" := "Drive 4 RUN FWD", "Drive Ready Signal" := "Drive 4 Ready", DelayTime :=, "Timer ET" =>, "Ouput WORD" => "Alarms".AlarmStruct.Alarm_Drive4)
   END_RUNG
   // the same network as SCL:
   "DriveConfirmation_Function_Axis 4"("System RUN" := "Systeem RUN",   // "DriveConfirmation_Function"
                           "Drive Ouput Q" := "Drive 4 RUN FWD",
                           "Drive Ready Signal" := "Drive 4 Ready",
                           "Ouput WORD" => "Alarms".AlarmStruct.Alarm_Drive4);
END_REGION

REGION Network 21: Confirmation Drive 5
   RUNG wire#powerrail
      "DriveConfirmation_Function_Axis 5"("System RUN" := "Systeem RUN", "Drive Ouput Q" := "Drive 5 RUN FWD", "Drive Ready Signal" := "Drive 5 Ready", DelayTime :=, "Timer ET" =>, "Ouput WORD" => "Alarms".AlarmStruct.Alarm_Drive5)
   END_RUNG
   // the same network as SCL:
   "DriveConfirmation_Function_Axis 5"("System RUN" := "Systeem RUN",   // "DriveConfirmation_Function"
                           "Drive Ouput Q" := "Drive 5 RUN FWD",
                           "Drive Ready Signal" := "Drive 5 Ready",
                           "Ouput WORD" => "Alarms".AlarmStruct.Alarm_Drive5);
END_REGION

REGION Network 22: EnoughProducts_OnInfeed
   RUNG wire#powerrail
      Contact( "Systeem RUN" )
      Contact( "NotEnoughProducts".Q )
      Coil( #EnoughProductsOnInfeed )
   END_RUNG
   // the same network as SCL:
   #EnoughProductsOnInfeed := "Systeem RUN" AND "NotEnoughProducts".Q;
END_REGION

REGION Network 23: NotEnoughProducts_OnInfeed
   RUNG wire#powerrail
      Contact( "Systeem RUN" )
      I_Contact( "Sensor Op Band" )
      { S7_Templates := "time_type := Time" } "NotEnoughProducts".TON(pt := "PLCMemory".InfeedTimeOutPT, et =>)
      Coil( #NotEnoughProductsOnInfeed )
   END_RUNG
   // the same network as SCL:
   "NotEnoughProducts".TON(IN := "Systeem RUN" AND NOT "Sensor Op Band", PT := "PLCMemory".InfeedTimeOutPT);
   #NotEnoughProductsOnInfeed := "NotEnoughProducts".Q;
END_REGION

REGION Network 24: RS Warning Not Enough Products
   RUNG wire#powerrail
      Contact( "Reset Active" )
      S_RS(operand := #Warning_NotEnoughProducts, s1 := #NotEnoughProductsOnInfeed)
      Coil( #TurnOffDrives )
   END_RUNG
   // the same network as SCL:
   IF "Reset Active" THEN
       #Warning_NotEnoughProducts := FALSE;   // RS flip-flop
   END_IF;
   IF #NotEnoughProductsOnInfeed THEN #Warning_NotEnoughProducts := TRUE; END_IF;
   #TurnOffDrives := #Warning_NotEnoughProducts;
END_REGION

REGION Network 25: TurnOff Drives Bypass
   RUNG wire#powerrail
      Contact( #TurnOffDrives )
      I_Contact( "TurnOff_InfeedTimeout" )
      Coil( "TurnOffDrive2" )
      Coil( "TurnOffDrive4" )
   END_RUNG
   // the same network as SCL:
   "TurnOffDrive2" := #TurnOffDrives AND NOT "TurnOff_InfeedTimeout";
   "TurnOffDrive4" := "TurnOffDrive2";
END_REGION
END_FUNCTION

FUNCTION_BLOCK "ESB_Flash_Warning_Block"   // FB1, FBD
VERSION : 0.1
// stored: AutoNumber true, IsIECCheckEnabled false, UDAEnableTagReadback false
   VAR_INPUT
      "Safety Feedback Contact" : Bool;
      "WarningTimer Time 1" : Time := T#150ms;
      "WarningTimer Time 2" : Time := T#150ms;
   END_VAR
   VAR_OUTPUT
      "Warning Ouput Contact" : Bool;
      "ET WarningTimer 1" : Time;
      "ET WarningTimer 2" : Time;
   END_VAR
   VAR_TEMP
      SafetyTakeoverContact : Bool;
   END_VAR
   VAR_TEMP   // added for the SCL form of the ladder/FBD networks
      _w1 : Bool;
   END_VAR
BEGIN

REGION Network 1: Flash Warning
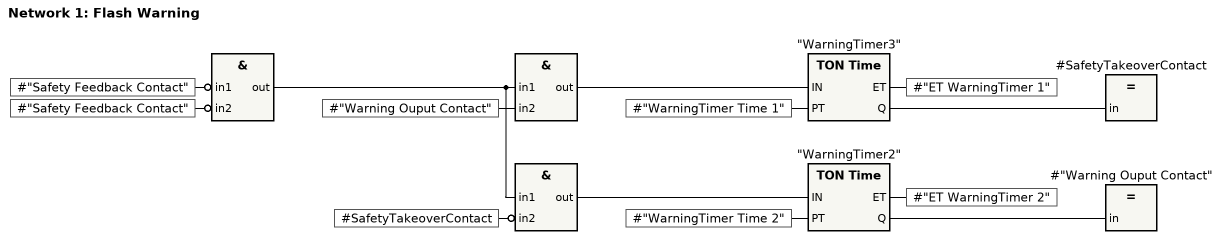
   #_w1 := NOT #"Safety Feedback Contact" AND NOT #"Safety Feedback Contact";
   "WarningTimer3".TON(IN := #_w1 AND #"Warning Ouput Contact",
                       PT := #"WarningTimer Time 1",
                       ET => #"ET WarningTimer 1");
   #SafetyTakeoverContact := "WarningTimer3".Q;
   "WarningTimer2".TON(IN := #_w1 AND NOT #SafetyTakeoverContact,
                       PT := #"WarningTimer Time 2",
                       ET => #"ET WarningTimer 2");
   #"Warning Ouput Contact" := "WarningTimer2".Q;
END_REGION
END_FUNCTION_BLOCK

FUNCTION_BLOCK "Delayed_Message_Function"   // FB2, FBD
TITLE = Delayed Message Function
VERSION : 0.1
// Functionblock For Delaying Message Function for example for filling an magazine or waiting for an signal. It is possible to adjust Time with the Dleay Time Message Input. The FlashTimer Time 1 & 2 ar for adjusting the flashing time of the ouput LED.
// stored: AutoNumber true, IsIECCheckEnabled false, UDAEnableTagReadback false
   VAR_INPUT
      "Override Message" : Bool;
      "Sensor Input 1" : Bool;
      "Sensor Input 2" : Bool := true;
      "Delay Time Message" : Time := T#1S_500MS;
      "FlashTimer Time 1" : Time := T#200ms;
      "FlashTimer Time 2" : Time := T#200ms;
   END_VAR
   VAR_OUTPUT
      "Output Signal" : Bool;
      "Output Signal Halt" : Bool;
      "ET Delayed Timer" : Time;
      "Output LED Flashing" : Bool;
   END_VAR
   VAR_TEMP
      "Internal Delayed Signal" : Bool;
   END_VAR
   VAR_TEMP   // added for the SCL form of the ladder/FBD networks
      _w1 : Bool;
   END_VAR
BEGIN

REGION Network 1: Delayed Signal to Outputs
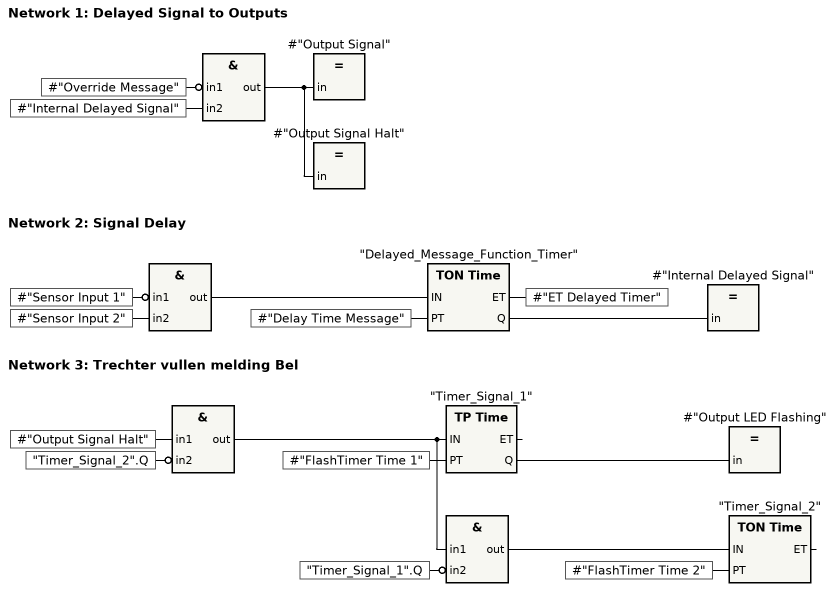
   #"Output Signal" := NOT #"Override Message" AND #"Internal Delayed Signal";
   #"Output Signal Halt" := #"Output Signal";
END_REGION

REGION Network 2: Signal Delay
   "Delayed_Message_Function_Timer".TON(IN := NOT #"Sensor Input 1" AND #"Sensor Input 2",
                           PT := #"Delay Time Message",
                           ET => #"ET Delayed Timer");
   #"Internal Delayed Signal" := "Delayed_Message_Function_Timer".Q;
END_REGION

REGION Network 3: Trechter vullen melding Bel
   #_w1 := #"Output Signal Halt" AND NOT "Timer_Signal_2".Q;
   "Timer_Signal_1".TP(IN := #_w1, PT := #"FlashTimer Time 1");
   #"Output LED Flashing" := "Timer_Signal_1".Q;
   "Timer_Signal_2".TON(IN := #_w1 AND NOT "Timer_Signal_1".Q, PT := #"FlashTimer Time 2");
END_REGION
END_FUNCTION_BLOCK

FUNCTION_BLOCK "Alarm_Axis_Position_Function"   // FB3, FBD
TITLE = Alarm Axis not in Position
VERSION : 0.1
// stored: AutoNumber true, IsIECCheckEnabled false, UDAEnableTagReadback false
   VAR_INPUT
      "Axis FWD command" : Bool;
      "Axis Feedback (Sensor) signal" : Bool;
      "Axis Encoder Singal" : Real;
      "Axis Command Position" : Real;
      "Sensor Controlled (HIGH) - Position Controlled (LOW)" : Bool;
      "CheckTime Setting" : Time := T#5S;
   END_VAR
   VAR_OUTPUT
      "Alarm BOOL" : Bool;
      "Alarm WORD" : Bool;
   END_VAR
   VAR_TEMP
      "Axis Feedback Internal" : Bool;
      "Axis Encoder On Position" : Bool;
      "Axis Sensor On Position" : Bool;
      "Axis Measuring Mode" : Bool;
   END_VAR
BEGIN

REGION Network 1: When axis is spinning start timer
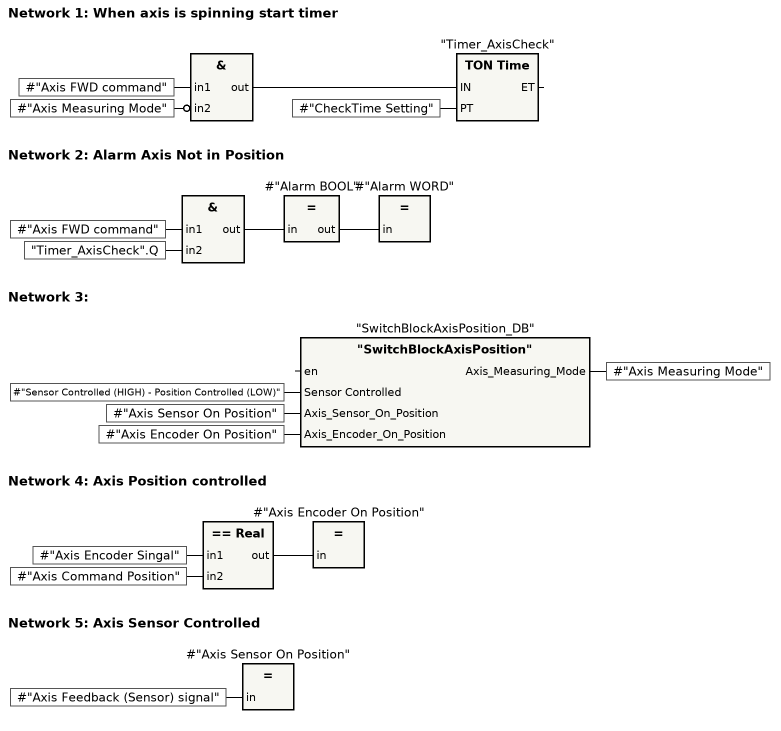
   "Timer_AxisCheck".TON(IN := #"Axis FWD command" AND NOT #"Axis Measuring Mode", PT := #"CheckTime Setting");
END_REGION

REGION Network 2: Alarm Axis Not in Position
   #"Alarm BOOL" := #"Axis FWD command" AND "Timer_AxisCheck".Q;
   #"Alarm WORD" := #"Alarm BOOL";
END_REGION

REGION Network 3
   "SwitchBlockAxisPosition_DB"("Sensor Controlled" := #"Sensor Controlled (HIGH) - Position Controlled (LOW)",   // "SwitchBlockAxisPosition"
                           Axis_Sensor_On_Position := #"Axis Sensor On Position",
                           Axis_Encoder_On_Position := #"Axis Encoder On Position",
                           Axis_Measuring_Mode => #"Axis Measuring Mode");
END_REGION

REGION Network 4: Axis Position controlled
   #"Axis Encoder On Position" := #"Axis Encoder Singal" = #"Axis Command Position";
END_REGION

REGION Network 5: Axis Sensor Controlled
   #"Axis Sensor On Position" := #"Axis Feedback (Sensor) signal";
END_REGION
END_FUNCTION_BLOCK

FUNCTION_BLOCK "SwitchBlockAxisPosition"
{ S7_Optimized_Access := 'FALSE' }
VERSION : 0.1
   VAR_INPUT 
      "Sensor Controlled" : Bool;
      Axis_Sensor_On_Position : Bool;
      Axis_Encoder_On_Position : Bool;
   END_VAR

   VAR_OUTPUT 
      Axis_Measuring_Mode : Bool;
   END_VAR


BEGIN
	IF #"Sensor Controlled" THEN
	    #Axis_Measuring_Mode := #Axis_Sensor_On_Position;
	ELSE
	    #Axis_Measuring_Mode := #Axis_Encoder_On_Position;
	END_IF;
	
END_FUNCTION_BLOCK

FUNCTION_BLOCK "DriveConfirmation_Function"   // FB5, FBD
TITLE = Drive Confirmation Function Block
VERSION : 0.1
// stored: AutoNumber true, IsIECCheckEnabled false, UDAEnableTagReadback false
   VAR_INPUT
      "System RUN" : Bool;
      "Drive Ouput Q" : Bool;
      "Drive Ready Signal" : Bool;
      DelayTime : Time := T#1s;
   END_VAR
   VAR_OUTPUT
      "Timer ET" : Time;
      "Ouput WORD" : Bool;
   END_VAR
BEGIN

REGION Network 1: Confirmation Drive
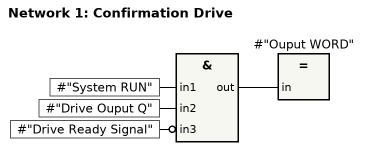
   #"Ouput WORD" := #"System RUN" AND #"Drive Ouput Q" AND NOT #"Drive Ready Signal";
END_REGION
END_FUNCTION_BLOCK

FUNCTION "9 - OVERIG" : Void   // FC6, LAD
TITLE = Other - Testing
VERSION : 0.1
// stored: AutoNumber true, IsIECCheckEnabled false, UDAEnableTagReadback false
   VAR_TEMP
      Encoder : Int;
      Gate : Bool;
      GATESTP : Bool;
      OTERRA : Bool;
      Direct : Bool;
      Prepar : Bool;
      CMPV1 : Bool;
      CMPV2 : Bool;
      RESSYNC : Bool;
      RESZERO : Bool;
      OTERR : Bool;
   END_VAR
BEGIN

REGION Network 1: SAFETY - OVERRIDE
